LIN {X 0,Y 197.924,Z 366.595,A -85,B 0,C 180,E1 -22444.008,E2 -22444.008} C_VEL
LIN {X 0,Y 203.129,Z 358.179,A -85,B 0,C 180,E1 -22446.646,E2 -22446.646} C_VEL
LIN {X 0,Y 207.879,Z 349.395,A -85,B 0,C 180,E1 -22448.886,E2 -22448.886} C_VEL
LIN {X 0,Y 213.116,Z 339.014,A -85,B 0,C 180,E1 -22450.955,E2 -22450.955} C_VEL
LIN {X 0,Y 218.33,Z 327.013,A -85,B 0,C 180,E1 -22452.848,E2 -22452.848} C_VEL
LIN {X 0,Y 222.672,Z 315.199,A -85,B 0,C 180,E1 -22454.295,E2 -22454.295} C_VEL
LIN {X 0,Y 226.681,Z 302.215,A -85,B 0,C 180,E1 -22455.49,E2 -22455.49} C_VEL
LIN {X 0,Y 230.05,Z 288.122,A -85,B 0,C 180,E1 -22456.439,E2 -22456.439} C_VEL
LIN {X 0,Y 232.521,Z 273.354,A -85,B 0,C 180,E1 -22457.126,E2 -22457.126} C_VEL
LIN {X 0,Y 234.238,Z 254.152,A -85,B 0,C 180,E1 -22457.708,E2 -22457.708} C_VEL
LIN {X 0,Y 236.836,Z 218.214,A -85,B 0,C 180,E1 -22458.708,E2 -22458.708} C_VEL
LIN {X 0,Y 232.194,Z 207.283,A -85,B 0,C 180,E1 -22461.02,E2 -22461.02} C_VEL
LIN {X 0,Y 227.459,Z 197.713,A -85,B 0,C 180,E1 -22463.554,E2 -22463.554} C_VEL
LIN {X 0,Y 222.962,Z 189.346,A -85,B 0,C 180,E1 -22466.218,E2 -22466.218} C_VEL
LIN {X 0,Y 219.708,Z 183.706,A -85,B 0,C 180,E1 -22468.352,E2 -22468.352} C_VEL
LIN {X 0,Y 216.874,Z 179.005,A -85,B 0,C 180,E1 -22470.433,E2 -22470.433} C_VEL
LIN {X 0,Y 214.738,Z 175.538,A -85,B 0,C 180,E1 -22472.178,E2 -22472.178} C_VEL
LIN {X 0,Y 211.845,Z 170.966,A -85,B 0,C 180,E1 -22474.848,E2 -22474.848} C_VEL
LIN {X 0,Y 209.156,Z 167.545,A -85,B 0,C 180,E1 -22477.703,E2 -22477.703} C_VEL
LIN {X 0,Y 207.226,Z 164.238,A -85,B 0,C 180,E1 -22480.325,E2 -22480.325} C_VEL
LIN {X 0,Y 203.698,Z 160.294,A -85,B 0,C 180,E1 -22488.046,E2 -22488.046} C_VEL
LIN {X 0,Y 203.417,Z 158.582,A -85,B 0,C 180,E1 -22490.606,E2 -22490.606} C_VEL
LIN {X 0,Y 203.441,Z 158.596,A -85,B 0,C 180,E1 -22494.045,E2 -22494.045} C_VEL
LIN {X 0,Y 204.542,Z 161.074,A -85,B 0,C 180,E1 -22499.009,E2 -22499.009} C_VEL
LIN {X 0,Y 206.776,Z 163.712,A -85,B 0,C 180,E1 -22503.403,E2 -22503.403} C_VEL
LIN {X 0,Y 207.532,Z 164.297,A -85,B 0,C 180,E1 -22504.485,E2 -22504.485} C_VEL
LIN {X 0,Y 209.461,Z 167.504,A -85,B 0,C 180,E1 -22507.018,E2 -22507.018} C_VEL
LIN {X 0,Y 211.323,Z 169.48,A -85,B 0,C 180,E1 -22508.967,E2 -22508.967} C_VEL
LIN {X 0,Y 213.7,Z 172.996,A -85,B 0,C 180,E1 -22511.242,E2 -22511.242} C_VEL
LIN {X 0,Y 215.003,Z 174.469,A -85,B 0,C 180,E1 -22512.327,E2 -22512.327} C_VEL
LIN {X 0,Y 218.65,Z 179.753,A -85,B 0,C 180,E1 -22515.145,E2 -22515.145} C_VEL
LIN {X 0,Y 221.807,Z 184.294,A -85,B 0,C 180,E1 -22517.249,E2 -22517.249} C_VEL
LIN {X 0,Y 225.031,Z 189.073,A -85,B 0,C 180,E1 -22519.193,E2 -22519.193} C_VEL
LIN {X 0,Y 229.645,Z 196.427,A -85,B 0,C 180,E1 -22521.724,E2 -22521.724} C_VEL
LIN {X 0,Y 234.735,Z 206.452,A -85,B 0,C 180,E1 -22524.318,E2 -22524.318} C_VEL
LIN {X 0,Y 237.327,Z 212.29,A -85,B 0,C 180,E1 -22525.571,E2 -22525.571} C_VEL
LIN {X 0,Y 233.316,Z 263.334,A -85,B 0,C 180,E1 -22526.974,E2 -22526.974} C_VEL
LIN {X 0,Y 231.099,Z 278.043,A -85,B 0,C 180,E1 -22527.649,E2 -22527.649} C_VEL
LIN {X 0,Y 228.064,Z 291.816,A -85,B 0,C 180,E1 -22528.563,E2 -22528.563} C_VEL
LIN {X 0,Y 224.528,Z 304.669,A -85,B 0,C 180,E1 -22529.768,E2 -22529.768} C_VEL
LIN {X 0,Y 220.106,Z 317.534,A -85,B 0,C 180,E1 -22531.332,E2 -22531.332} C_VEL
LIN {X 0,Y 215.155,Z 329.395,A -85,B 0,C 180,E1 -22533.168,E2 -22533.168} C_VEL
LIN {X 0,Y 210.454,Z 339.175,A -85,B 0,C 180,E1 -22535.094,E2 -22535.094} C_VEL
LIN {X 0,Y 205.546,Z 348.318,A -85,B 0,C 180,E1 -22537.344,E2 -22537.344} C_VEL
LIN {X 0,Y 200.059,Z 357.453,A -85,B 0,C 180,E1 -22540.172,E2 -22540.172} C_VEL
LIN {X 0,Y 194.996,Z 365.083,A -85,B 0,C 180,E1 -22543.208,E2 -22543.208} C_VEL
LIN {X 0,Y 190,Z 372.03,A -85,B 0,C 180,E1 -22546.815,E2 -22546.815} C_VEL
LIN {X 0,Y 186.208,Z 376.82,A -85,B 0,C 180,E1 -22550.083,E2 -22550.083} C_VEL
LIN {X 0,Y 182.741,Z 380.951,A -85,B 0,C 180,E1 -22553.85,E2 -22553.85} C_VEL
LIN {X 0,Y 180.515,Z 383.439,A -85,B 0,C 180,E1 -22556.967,E2 -22556.967} C_VEL
LIN {X 0,Y 177.978,Z 385.836,A -85,B 0,C 180,E1 -22561.712,E2 -22561.712} C_VEL
LIN {X 0,Y 176.489,Z 386.756,A -85,B 0,C 180,E1 -22566.53,E2 -22566.53} C_VEL
LIN {X 0,Y 175.717,Z 386.244,A -85,B 0,C 180,E1 -22571.336,E2 -22571.336} C_VEL
LIN {X 0,Y 175.641,Z 385.441,A -85,B 0,C 180,E1 -22573.772,E2 -22573.772} C_VEL
LIN {X 0,Y 175.765,Z 382.819,A -85,B 0,C 180,E1 -22578.464,E2 -22578.464} C_VEL
LIN {X 0,Y 176.339,Z 379.84,A -85,B 0,C 180,E1 -22581.978,E2 -22581.978} C_VEL
LIN {X 0,Y 177.183,Z 376.025,A -85,B 0,C 180,E1 -22585.447,E2 -22585.447} C_VEL
LIN {X 0,Y 178.317,Z 371.31,A -85,B 0,C 180,E1 -22588.868,E2 -22588.868} C_VEL
LIN {X 0,Y 180.274,Z 364.443,A -85,B 0,C 180,E1 -22592.79,E2 -22592.79} C_VEL
LIN {X 0,Y 182.883,Z 355.918,A -85,B 0,C 180,E1 -22596.617,E2 -22596.617} C_VEL
LIN {X 0,Y 185.69,Z 346.926,A -85,B 0,C 180,E1 -22599.834,E2 -22599.834} C_VEL
LIN {X 0,Y 188.154,Z 338.243,A -85,B 0,C 180,E1 -22602.399,E2 -22602.399} C_VEL
LIN {X 0,Y 190.884,Z 328.903,A -85,B 0,C 180,E1 -22604.659,E2 -22604.659} C_VEL
LIN {X 0,Y 193.795,Z 317.727,A -85,B 0,C 180,E1 -22606.862,E2 -22606.862} C_VEL
LIN {X 0,Y 196.622,Z 305.546,A -85,B 0,C 180,E1 -22608.762,E2 -22608.762} C_VEL
LIN {X 0,Y 199.012,Z 293.194,A -85,B 0,C 180,E1 -22610.272,E2 -22610.272} C_VEL
LIN {X 0,Y 201.044,Z 279.549,A -85,B 0,C 180,E1 -22611.531,E2 -22611.531} C_VEL
LIN {X 0,Y 202.585,Z 265.477,A -85,B 0,C 180,E1 -22612.43,E2 -22612.43} C_VEL
LIN {X 0,Y 203.759,Z 246.646,A -85,B 0,C 180,E1 -22613.151,E2 -22613.151} C_VEL
LIN {X 0,Y 207.071,Z 187.142,A -85,B 0,C 180,E1 -22615.036,E2 -22615.036} C_VEL
LIN {X 0,Y 202.861,Z 176.015,A -85,B 0,C 180,E1 -22616.361,E2 -22616.361} C_VEL
LIN {X 0,Y 196.456,Z 163.46,A -85,B 0,C 180,E1 -22618.321,E2 -22618.321} C_VEL
LIN {X 0,Y 188.904,Z 150.475,A -85,B 0,C 180,E1 -22620.783,E2 -22620.783} C_VEL
LIN {X 0,Y 183.421,Z 142.139,A -85,B 0,C 180,E1 -22622.704,E2 -22622.704} C_VEL
LIN {X 0,Y 180.927,Z 138.404,A -85,B 0,C 180,E1 -22623.626,E2 -22623.626} C_VEL
LIN {X 0,Y 179.099,Z 136.063,A -85,B 0,C 180,E1 -22624.304,E2 -22624.304} C_VEL
LIN {X 0,Y 178.464,Z 133.88,A -85,B 0,C 180,E1 -22624.658,E2 -22624.658} C_VEL
LIN {X 0,Y 178.477,Z 133.875,A -85,B 0,C 180,E1 -22629.049,E2 -22629.049} C_VEL
LIN {X 0,Y 178.494,Z 133.859,A -85,B 0,C 180,E1 -22632.013,E2 -22632.013} C_VEL
LIN {X 0,Y 178.504,Z 133.854,A -85,B 0,C 180,E1 -22635.123,E2 -22635.123} C_VEL
LIN {X 0,Y 178.493,Z 133.87,A -85,B 0,C 180,E1 -22638.421,E2 -22638.421} C_VEL
LIN {X 0,Y 178.444,Z 133.86,A -85,B 0,C 180,E1 -22643.799,E2 -22643.799} C_VEL
LIN {X 0,Y 178.466,Z 133.878,A -85,B 0,C 180,E1 -22646.553,E2 -22646.553} C_VEL
LIN {X 0,Y 178.499,Z 133.842,A -85,B 0,C 180,E1 -22650.013,E2 -22650.013} C_VEL
LIN {X 0,Y 178.525,Z 133.862,A -85,B 0,C 180,E1 -22654.875,E2 -22654.875} C_VEL
LIN {X 0,Y 178.638,Z 133.852,A -85,B 0,C 180,E1 -22660.761,E2 -22660.761} C_VEL
LIN {X 0,Y 178.663,Z 133.849,A -85,B 0,C 180,E1 -22664.025,E2 -22664.025} C_VEL
LIN {X 0,Y 178.88,Z 133.825,A -85,B 0,C 180,E1 -22669.161,E2 -22669.161} C_VEL
LIN {X 0,Y 178.918,Z 133.782,A -85,B 0,C 180,E1 -22673.24,E2 -22673.24} C_VEL
LIN {X 0,Y 179.146,Z 133.788,A -85,B 0,C 180,E1 -22677.759,E2 -22677.759} C_VEL
LIN {X 0,Y 179.363,Z 133.764,A -85,B 0,C 180,E1 -22680.007,E2 -22680.007} C_VEL
LIN {X 0,Y 178.863,Z 133.791,A -85,B 0,C 180,E1 -22684.515,E2 -22684.515} C_VEL
LIN {X 0,Y 178.953,Z 133.817,A -85,B 0,C 180,E1 -22689.045,E2 -22689.045} C_VEL
LIN {X 0,Y 178.682,Z 133.85,A -85,B 0,C 180,E1 -22693.657,E2 -22693.657} C_VEL
LIN {X 0,Y 178.647,Z 133.853,A -85,B 0,C 180,E1 -22698.351,E2 -22698.351} C_VEL
LIN {X 0,Y 178.51,Z 133.872,A -85,B 0,C 180,E1 -22703.192,E2 -22703.192} C_VEL
LIN {X 0,Y 178.487,Z 133.863,A -85,B 0,C 180,E1 -22708.204,E2 -22708.204} C_VEL
LIN {X 0,Y 178.479,Z 133.872,A -85,B 0,C 180,E1 -22710.798,E2 -22710.798} C_VEL
LIN {X 0,Y 178.486,Z 133.875,A -85,B 0,C 180,E1 -22714.226,E2 -22714.226} C_VEL
LIN {X 0,Y 178.411,Z 134.02,A -85,B 0,C 180,E1 -22719,E2 -22719} C_VEL
LIN {X 0,Y 179.403,Z 136.688,A -85,B 0,C 180,E1 -22719.454,E2 -22719.454} C_VEL
LIN {X 0,Y 181.505,Z 139.246,A -85,B 0,C 180,E1 -22720.224,E2 -22720.224} C_VEL
LIN {X 0,Y 183.847,Z 142.743,A -85,B 0,C 180,E1 -22721.083,E2 -22721.083} C_VEL
LIN {X 0,Y 187.701,Z 149.384,A -85,B 0,C 180,E1 -22722.472,E2 -22722.472} C_VEL
LIN {X 0,Y 194.053,Z 161.878,A -85,B 0,C 180,E1 -22724.674,E2 -22724.674} C_VEL
LIN {X 0,Y 199.515,Z 174.348,A -85,B 0,C 180,E1 -22726.489,E2 -22726.489} C_VEL
LIN {X 0,Y 206.104,Z 192.069,A -85,B 0,C 180,E1 -22728.614,E2 -22728.614} C_VEL
LIN {X 0,Y 206.705,Z 198.43,A -85,B 0,C 180,E1 -22728.999,E2 -22728.999} C_VEL
LIN {X 0,Y 204.554,Z 239.005,A -85,B 0,C 180,E1 -22730.303,E2 -22730.303} C_VEL
LIN {X 0,Y 203.706,Z 244.85,A -85,B 0,C 180,E1 -22730.389,E2 -22730.389} C_VEL
LIN {X 0,Y 197.796,Z 263.79,A -85,B 0,C 180,E1 -22730.093,E2 -22730.093} C_VEL
LIN {X 0,Y 196.896,Z 269.616,A -85,B 0,C 180,E1 -22730.218,E2 -22730.218} C_VEL
LIN {X 0,Y 195.425,Z 283.938,A -85,B 0,C 180,E1 -22731.002,E2 -22731.002} C_VEL
LIN {X 0,Y 193.265,Z 297.901,A -85,B 0,C 180,E1 -22732.15,E2 -22732.15} C_VEL
LIN {X 0,Y 190.76,Z 310.487,A -85,B 0,C 180,E1 -22733.557,E2 -22733.557} C_VEL
LIN {X 0,Y 188.351,Z 320.636,A -85,B 0,C 180,E1 -22734.997,E2 -22734.997} C_VEL
LIN {X 0,Y 185.153,Z 333.155,A -85,B 0,C 180,E1 -22737.259,E2 -22737.259} C_VEL
LIN {X 0,Y 182.733,Z 341.231,A -85,B 0,C 180,E1 -22739.046,E2 -22739.046} C_VEL
LIN {X 0,Y 179.902,Z 350.234,A -85,B 0,C 180,E1 -22741.413,E2 -22741.413} C_VEL
LIN {X 0,Y 176.695,Z 360.281,A -85,B 0,C 180,E1 -22744.69,E2 -22744.69} C_VEL
LIN {X 0,Y 173.88,Z 369.292,A -85,B 0,C 180,E1 -22748.393,E2 -22748.393} C_VEL
LIN {X 0,Y 171.794,Z 376.544,A -85,B 0,C 180,E1 -22752.136,E2 -22752.136} C_VEL
LIN {X 0,Y 170.316,Z 382.067,A -85,B 0,C 180,E1 -22755.669,E2 -22755.669} C_VEL
LIN {X 0,Y 169.282,Z 387.851,A -85,B 0,C 180,E1 -22760.444,E2 -22760.444} C_VEL
LIN {X 0,Y 168.89,Z 392.01,A -85,B 0,C 180,E1 -22765.229,E2 -22765.229} C_VEL
LIN {X 0,Y 169.024,Z 394.686,A -85,B 0,C 180,E1 -22770.003,E2 -22770.003} C_VEL
LIN {X 0,Y 168.891,Z 395.944,A -85,B 0,C 180,E1 -22774.777,E2 -22774.777} C_VEL
LIN {X 0,Y 169.339,Z 395.878,A -85,B 0,C 180,E1 -22779.559,E2 -22779.559} C_VEL
LIN {X 0,Y 170.625,Z 394.512,A -85,B 0,C 180,E1 -22784.312,E2 -22784.312} C_VEL
LIN {X 0,Y 173.086,Z 391.826,A -85,B 0,C 180,E1 -22788.959,E2 -22788.959} C_VEL
LIN {X 0,Y 176.47,Z 387.752,A -85,B 0,C 180,E1 -22793.472,E2 -22793.472} C_VEL
LIN {X 0,Y 180.936,Z 382.174,A -85,B 0,C 180,E1 -22797.785,E2 -22797.785} C_VEL
LIN {X 0,Y 186.475,Z 374.921,A -85,B 0,C 180,E1 -22801.85,E2 -22801.85} C_VEL
LIN {X 0,Y 192.081,Z 366.957,A -85,B 0,C 180,E1 -22805.192,E2 -22805.192} C_VEL
LIN {X 0,Y 197.505,Z 358.65,A -85,B 0,C 180,E1 -22807.87,E2 -22807.87} C_VEL
LIN {X 0,Y 203.298,Z 348.508,A -85,B 0,C 180,E1 -22810.481,E2 -22810.481} C_VEL
LIN {X 0,Y 208.901,Z 337.643,A -85,B 0,C 180,E1 -22812.618,E2 -22812.618} C_VEL
LIN {X 0,Y 214.329,Z 325.298,A -85,B 0,C 180,E1 -22814.503,E2 -22814.503} C_VEL
LIN {X 0,Y 218.881,Z 313.11,A -85,B 0,C 180,E1 -22815.929,E2 -22815.929} C_VEL
LIN {X 0,Y 223.002,Z 299.6,A -85,B 0,C 180,E1 -22817.119,E2 -22817.119} C_VEL
LIN {X 0,Y 226.321,Z 285.451,A -85,B 0,C 180,E1 -22818.02,E2 -22818.02} C_VEL
LIN {X 0,Y 228.543,Z 271.735,A -85,B 0,C 180,E1 -22818.627,E2 -22818.627} C_VEL
LIN {X 0,Y 231.009,Z 242.939,A -85,B 0,C 180,E1 -22819.448,E2 -22819.448} C_VEL
LIN {X 0,Y 232.645,Z 221.01,A -85,B 0,C 180,E1 -22820.066,E2 -22820.066} C_VEL
LIN {X 0,Y 228.5,Z 211.213,A -85,B 0,C 180,E1 -22822.271,E2 -22822.271} C_VEL
LIN {X 0,Y 224.543,Z 202.944,A -85,B 0,C 180,E1 -22824.528,E2 -22824.528} C_VEL
LIN {X 0,Y 220.56,Z 195.258,A -85,B 0,C 180,E1 -22827.022,E2 -22827.022} C_VEL
LIN {X 0,Y 217.491,Z 189.717,A -85,B 0,C 180,E1 -22829.15,E2 -22829.15} C_VEL
LIN {X 0,Y 213.44,Z 182.601,A -85,B 0,C 180,E1 -22832.427,E2 -22832.427} C_VEL
LIN {X 0,Y 210.315,Z 177.667,A -85,B 0,C 180,E1 -22835.394,E2 -22835.394} C_VEL
LIN {X 0,Y 207.948,Z 174.459,A -85,B 0,C 180,E1 -22838.019,E2 -22838.019} C_VEL
LIN {X 0,Y 205.85,Z 170.917,A -85,B 0,C 180,E1 -22841.018,E2 -22841.018} C_VEL
LIN {X 0,Y 202.767,Z 167.321,A -85,B 0,C 180,E1 -22848.244,E2 -22848.244} C_VEL
LIN {X 0,Y 202.501,Z 165.535,A -85,B 0,C 180,E1 -22851.124,E2 -22851.124} C_VEL
LIN {X 0,Y 202.572,Z 165.825,A -85,B 0,C 180,E1 -22854.283,E2 -22854.283} C_VEL
LIN {X 0,Y 203.553,Z 168.062,A -85,B 0,C 180,E1 -22858.757,E2 -22858.757} C_VEL
LIN {X 0,Y 205.721,Z 170.676,A -85,B 0,C 180,E1 -22863.176,E2 -22863.176} C_VEL
LIN {X 0,Y 206.358,Z 171.324,A -85,B 0,C 180,E1 -22864.144,E2 -22864.144} C_VEL
LIN {X 0,Y 208.446,Z 174.671,A -85,B 0,C 180,E1 -22866.938,E2 -22866.938} C_VEL
LIN {X 0,Y 209.825,Z 176.191,A -85,B 0,C 180,E1 -22868.426,E2 -22868.426} C_VEL
LIN {X 0,Y 212.302,Z 179.809,A -85,B 0,C 180,E1 -22870.871,E2 -22870.871} C_VEL
LIN {X 0,Y 213.441,Z 181.322,A -85,B 0,C 180,E1 -22871.869,E2 -22871.869} C_VEL
LIN {X 0,Y 216.744,Z 186.164,A -85,B 0,C 180,E1 -22874.517,E2 -22874.517} C_VEL
LIN {X 0,Y 220.321,Z 191.498,A -85,B 0,C 180,E1 -22876.996,E2 -22876.996} C_VEL
LIN {X 0,Y 224.965,Z 198.794,A -85,B 0,C 180,E1 -22879.812,E2 -22879.812} C_VEL
LIN {X 0,Y 227.785,Z 203.912,A -85,B 0,C 180,E1 -22881.397,E2 -22881.397} C_VEL
LIN {X 0,Y 231.774,Z 212.095,A -85,B 0,C 180,E1 -22883.514,E2 -22883.514} C_VEL
LIN {X 0,Y 233.145,Z 215.09,A -85,B 0,C 180,E1 -22884.208,E2 -22884.208} C_VEL
LIN {X 0,Y 229.221,Z 263.339,A -85,B 0,C 180,E1 -22885.54,E2 -22885.54} C_VEL
LIN {X 0,Y 227.005,Z 277.668,A -85,B 0,C 180,E1 -22886.183,E2 -22886.183} C_VEL
LIN {X 0,Y 223.96,Z 291.248,A -85,B 0,C 180,E1 -22887.069,E2 -22887.069} C_VEL
LIN {X 0,Y 220.053,Z 304.97,A -85,B 0,C 180,E1 -22888.342,E2 -22888.342} C_VEL
LIN {X 0,Y 215.706,Z 317.209,A -85,B 0,C 180,E1 -22889.828,E2 -22889.828} C_VEL
LIN {X 0,Y 210.586,Z 329.163,A -85,B 0,C 180,E1 -22891.672,E2 -22891.672} C_VEL
LIN {X 0,Y 205.053,Z 340.237,A -85,B 0,C 180,E1 -22893.865,E2 -22893.865} C_VEL
LIN {X 0,Y 199.374,Z 350.201,A -85,B 0,C 180,E1 -22896.413,E2 -22896.413} C_VEL
LIN {X 0,Y 193.442,Z 359.417,A -85,B 0,C 180,E1 -22899.458,E2 -22899.458} C_VEL
LIN {X 0,Y 188.337,Z 366.604,A -85,B 0,C 180,E1 -22902.52,E2 -22902.52} C_VEL
LIN {X 0,Y 183.112,Z 373.348,A -85,B 0,C 180,E1 -22906.298,E2 -22906.298} C_VEL
LIN {X 0,Y 179.21,Z 377.935,A -85,B 0,C 180,E1 -22909.675,E2 -22909.675} C_VEL
LIN {X 0,Y 175.978,Z 381.516,A -85,B 0,C 180,E1 -22913.194,E2 -22913.194} C_VEL
LIN {X 0,Y 174.174,Z 383.378,A -85,B 0,C 180,E1 -22915.601,E2 -22915.601} C_VEL
LIN {X 0,Y 171.368,Z 385.895,A -85,B 0,C 180,E1 -22920.515,E2 -22920.515} C_VEL
LIN {X 0,Y 169.591,Z 386.933,A -85,B 0,C 180,E1 -22925.514,E2 -22925.514} C_VEL
LIN {X 0,Y 168.69,Z 386.534,A -85,B 0,C 180,E1 -22930.528,E2 -22930.528} C_VEL
LIN {X 0,Y 168.56,Z 385.64,A -85,B 0,C 180,E1 -22933.496,E2 -22933.496} C_VEL
LIN {X 0,Y 168.611,Z 383.286,A -85,B 0,C 180,E1 -22937.967,E2 -22937.967} C_VEL
LIN {X 0,Y 169.155,Z 380.413,A -85,B 0,C 180,E1 -22941.635,E2 -22941.635} C_VEL
LIN {X 0,Y 170.001,Z 376.719,A -85,B 0,C 180,E1 -22945.254,E2 -22945.254} C_VEL
LIN {X 0,Y 171.156,Z 372.089,A -85,B 0,C 180,E1 -22948.82,E2 -22948.82} C_VEL
LIN {X 0,Y 173.133,Z 365.392,A -85,B 0,C 180,E1 -22952.905,E2 -22952.905} C_VEL
LIN {X 0,Y 175.802,Z 357.048,A -85,B 0,C 180,E1 -22956.885,E2 -22956.885} C_VEL
LIN {X 0,Y 178.897,Z 347.578,A -85,B 0,C 180,E1 -22960.443,E2 -22960.443} C_VEL
LIN {X 0,Y 181.767,Z 337.828,A -85,B 0,C 180,E1 -22963.411,E2 -22963.411} C_VEL
LIN {X 0,Y 184.659,Z 328.358,A -85,B 0,C 180,E1 -22965.731,E2 -22965.731} C_VEL
LIN {X 0,Y 187.723,Z 317.019,A -85,B 0,C 180,E1 -22967.988,E2 -22967.988} C_VEL
LIN {X 0,Y 190.645,Z 304.637,A -85,B 0,C 180,E1 -22969.934,E2 -22969.934} C_VEL
LIN {X 0,Y 193.38,Z 290.832,A -85,B 0,C 180,E1 -22971.587,E2 -22971.587} C_VEL
LIN {X 0,Y 195.342,Z 277.108,A -85,B 0,C 180,E1 -22972.82,E2 -22972.82} C_VEL
LIN {X 0,Y 196.867,Z 262.852,A -85,B 0,C 180,E1 -22973.677,E2 -22973.677} C_VEL
LIN {X 0,Y 200.885,Z 196.744,A -85,B 0,C 180,E1 -22975.858,E2 -22975.858} C_VEL
LIN {X 0,Y 201.212,Z 188.949,A -85,B 0,C 180,E1 -22976.135,E2 -22976.135} C_VEL
LIN {X 0,Y 197.357,Z 178.875,A -85,B 0,C 180,E1 -22977.409,E2 -22977.409} C_VEL
LIN {X 0,Y 191.075,Z 166.594,A -85,B 0,C 180,E1 -22979.443,E2 -22979.443} C_VEL
LIN {X 0,Y 184.097,Z 154.645,A -85,B 0,C 180,E1 -22981.856,E2 -22981.856} C_VEL
LIN {X 0,Y 177.132,Z 143.849,A -85,B 0,C 180,E1 -22984.475,E2 -22984.475} C_VEL
LIN {X 0,Y 174.957,Z 140.891,A -85,B 0,C 180,E1 -22985.334,E2 -22985.334} C_VEL
LIN {X 0,Y 174.114,Z 139.492,A -85,B 0,C 180,E1 -22985.691,E2 -22985.691} C_VEL
LIN {X 0,Y 172.15,Z 137.141,A -85,B 0,C 180,E1 -22986.492,E2 -22986.492} C_VEL
LIN {X 0,Y 171.41,Z 134.76,A -85,B 0,C 180,E1 -22986.954,E2 -22986.954} C_VEL
LIN {X 0,Y 171.434,Z 134.733,A -85,B 0,C 180,E1 -22992.46,E2 -22992.46} C_VEL
LIN {X 0,Y 171.432,Z 134.753,A -85,B 0,C 180,E1 -22997.549,E2 -22997.549} C_VEL
LIN {X 0,Y 171.417,Z 134.721,A -85,B 0,C 180,E1 -23002.06,E2 -23002.06} C_VEL
LIN {X 0,Y 171.395,Z 134.752,A -85,B 0,C 180,E1 -23007.798,E2 -23007.798} C_VEL
LIN {X 0,Y 171.426,Z 134.718,A -85,B 0,C 180,E1 -23010.54,E2 -23010.54} C_VEL
LIN {X 0,Y 171.453,Z 134.75,A -85,B 0,C 180,E1 -23015.81,E2 -23015.81} C_VEL
LIN {X 0,Y 171.594,Z 134.73,A -85,B 0,C 180,E1 -23020.882,E2 -23020.882} C_VEL
LIN {X 0,Y 171.599,Z 134.724,A -85,B 0,C 180,E1 -23025.783,E2 -23025.783} C_VEL
LIN {X 0,Y 171.894,Z 134.682,A -85,B 0,C 180,E1 -23030.596,E2 -23030.596} C_VEL
LIN {X 0,Y 171.814,Z 134.673,A -85,B 0,C 180,E1 -23035.315,E2 -23035.315} C_VEL
LIN {X 0,Y 172.325,Z 134.641,A -85,B 0,C 180,E1 -23040.008,E2 -23040.008} C_VEL
LIN {X 0,Y 171.812,Z 134.668,A -85,B 0,C 180,E1 -23044.7,E2 -23044.7} C_VEL
LIN {X 0,Y 171.883,Z 134.7,A -85,B 0,C 180,E1 -23049.421,E2 -23049.421} C_VEL
LIN {X 0,Y 171.605,Z 134.733,A -85,B 0,C 180,E1 -23054.232,E2 -23054.232} C_VEL
LIN {X 0,Y 171.542,Z 134.742,A -85,B 0,C 180,E1 -23059.57,E2 -23059.57} C_VEL
LIN {X 0,Y 171.469,Z 134.749,A -85,B 0,C 180,E1 -23065.624,E2 -23065.624} C_VEL
LIN {X 0,Y 171.442,Z 134.75,A -85,B 0,C 180,E1 -23070.594,E2 -23070.594} C_VEL
LIN {X 0,Y 171.391,Z 134.759,A -85,B 0,C 180,E1 -23076.674,E2 -23076.674} C_VEL
LIN {X 0,Y 172.273,Z 137.408,A -85,B 0,C 180,E1 -23077.185,E2 -23077.185} C_VEL
LIN {X 0,Y 174.601,Z 140.281,A -85,B 0,C 180,E1 -23078.138,E2 -23078.138} C_VEL
LIN {X 0,Y 176.859,Z 143.654,A -85,B 0,C 180,E1 -23079.056,E2 -23079.056} C_VEL
LIN {X 0,Y 181.273,Z 150.337,A -85,B 0,C 180,E1 -23080.752,E2 -23080.752} C_VEL
LIN {X 0,Y 187.224,Z 161.787,A -85,B 0,C 180,E1 -23082.972,E2 -23082.972} C_VEL
LIN {X 0,Y 193.134,Z 174.722,A -85,B 0,C 180,E1 -23085.065,E2 -23085.065} C_VEL
LIN {X 0,Y 199.773,Z 192.505,A -85,B 0,C 180,E1 -23087.355,E2 -23087.355} C_VEL
LIN {X 0,Y 200.578,Z 195.555,A -85,B 0,C 180,E1 -23087.658,E2 -23087.658} C_VEL
LIN {X 0,Y 200.842,Z 199.819,A -85,B 0,C 180,E1 -23087.9,E2 -23087.9} C_VEL
LIN {X 0,Y 196.896,Z 269.616,A -85,B 0,C 180,E1 -23090.218,E2 -23090.218} C_VEL
LIN {X 0,Y 195.922,Z 275.406,A -85,B 0,C 180,E1 -23090.387,E2 -23090.387} C_VEL
LIN {X 0,Y 192.489,Z 284.69,A -85,B 0,C 180,E1 -23090.5,E2 -23090.5} C_VEL
LIN {X 0,Y 188.597,Z 293.797,A -85,B 0,C 180,E1 -23090.762,E2 -23090.762} C_VEL
LIN {X 0,Y 186.917,Z 299.319,A -85,B 0,C 180,E1 -23091.172,E2 -23091.172} C_VEL
LIN {X 0,Y 184.148,Z 312.294,A -85,B 0,C 180,E1 -23092.713,E2 -23092.713} C_VEL
LIN {X 0,Y 181.138,Z 324.295,A -85,B 0,C 180,E1 -23094.576,E2 -23094.576} C_VEL
LIN {X 0,Y 178.365,Z 334.301,A -85,B 0,C 180,E1 -23096.525,E2 -23096.525} C_VEL
LIN {X 0,Y 175.977,Z 342.273,A -85,B 0,C 180,E1 -23098.391,E2 -23098.391} C_VEL
LIN {X 0,Y 172.398,Z 352.871,A -85,B 0,C 180,E1 -23101.384,E2 -23101.384} C_VEL
LIN {X 0,Y 169.237,Z 362.449,A -85,B 0,C 180,E1 -23104.812,E2 -23104.812} C_VEL
LIN {X 0,Y 166.629,Z 370.348,A -85,B 0,C 180,E1 -23108.338,E2 -23108.338} C_VEL
LIN {X 0,Y 164.425,Z 377.927,A -85,B 0,C 180,E1 -23112.594,E2 -23112.594} C_VEL
LIN {X 0,Y 163.006,Z 383.156,A -85,B 0,C 180,E1 -23116.286,E2 -23116.286} C_VEL
LIN {X 0,Y 162.227,Z 387.382,A -85,B 0,C 180,E1 -23120.025,E2 -23120.025} C_VEL
LIN {X 0,Y 161.946,Z 389.695,A -85,B 0,C 180,E1 -23122.523,E2 -23122.523} C_VEL
LIN {X 0,Y 161.814,Z 393.172,A -85,B 0,C 180,E1 -23127.514,E2 -23127.514} C_VEL
LIN {X 0,Y 161.934,Z 394.368,A -85,B 0,C 180,E1 -23130.004,E2 -23130.004} C_VEL
LIN {X 0,Y 161.81,Z 395.698,A -85,B 0,C 180,E1 -23134.987,E2 -23134.987} C_VEL
LIN {X 0,Y 162.326,Z 395.706,A -85,B 0,C 180,E1 -23139.976,E2 -23139.976} C_VEL
LIN {X 0,Y 163.709,Z 394.42,A -85,B 0,C 180,E1 -23144.93,E2 -23144.93} C_VEL
LIN {X 0,Y 166.338,Z 391.824,A -85,B 0,C 180,E1 -23149.759,E2 -23149.759} C_VEL
LIN {X 0,Y 169.94,Z 387.837,A -85,B 0,C 180,E1 -23154.432,E2 -23154.432} C_VEL
LIN {X 0,Y 174.677,Z 382.342,A -85,B 0,C 180,E1 -23158.873,E2 -23158.873} C_VEL
LIN {X 0,Y 180.486,Z 375.178,A -85,B 0,C 180,E1 -23163.038,E2 -23163.038} C_VEL
LIN {X 0,Y 186.339,Z 367.314,A -85,B 0,C 180,E1 -23166.447,E2 -23166.447} C_VEL
LIN {X 0,Y 191.977,Z 359.12,A -85,B 0,C 180,E1 -23169.164,E2 -23169.164} C_VEL
LIN {X 0,Y 197.774,Z 349.473,A -85,B 0,C 180,E1 -23171.726,E2 -23171.726} C_VEL
LIN {X 0,Y 203.783,Z 338.448,A -85,B 0,C 180,E1 -23173.956,E2 -23173.956} C_VEL
LIN {X 0,Y 209.379,Z 326.422,A -85,B 0,C 180,E1 -23175.85,E2 -23175.85} C_VEL
LIN {X 0,Y 214.066,Z 314.565,A -85,B 0,C 180,E1 -23177.276,E2 -23177.276} C_VEL
LIN {X 0,Y 218.601,Z 300.415,A -85,B 0,C 180,E1 -23178.55,E2 -23178.55} C_VEL
LIN {X 0,Y 222.027,Z 286.604,A -85,B 0,C 180,E1 -23179.44,E2 -23179.44} C_VEL
LIN {X 0,Y 224.423,Z 272.754,A -85,B 0,C 180,E1 -23180.072,E2 -23180.072} C_VEL
LIN {X 0,Y 226.373,Z 252.123,A -85,B 0,C 180,E1 -23180.688,E2 -23180.688} C_VEL
LIN {X 0,Y 228.588,Z 223.962,A -85,B 0,C 180,E1 -23181.469,E2 -23181.469} C_VEL
LIN {X 0,Y 225.133,Z 215.618,A -85,B 0,C 180,E1 -23183.437,E2 -23183.437} C_VEL
LIN {X 0,Y 221.106,Z 206.893,A -85,B 0,C 180,E1 -23185.908,E2 -23185.908} C_VEL
LIN {X 0,Y 217.495,Z 199.828,A -85,B 0,C 180,E1 -23188.341,E2 -23188.341} C_VEL
LIN {X 0,Y 213.873,Z 193.038,A -85,B 0,C 180,E1 -23191.153,E2 -23191.153} C_VEL
LIN {X 0,Y 211.177,Z 188.352,A -85,B 0,C 180,E1 -23193.54,E2 -23193.54} C_VEL
LIN {X 0,Y 208.172,Z 183.358,A -85,B 0,C 180,E1 -23196.654,E2 -23196.654} C_VEL
LIN {X 0,Y 204.661,Z 177.829,A -85,B 0,C 180,E1 -23201.448,E2 -23201.448} C_VEL
LIN {X 0,Y 201.755,Z 174.043,A -85,B 0,C 180,E1 -23208.948,E2 -23208.948} C_VEL
LIN {X 0,Y 201.611,Z 172.649,A -85,B 0,C 180,E1 -23211.085,E2 -23211.085} C_VEL
LIN {X 0,Y 201.658,Z 172.794,A -85,B 0,C 180,E1 -23213.992,E2 -23213.992} C_VEL
LIN {X 0,Y 202.581,Z 175.069,A -85,B 0,C 180,E1 -23218.548,E2 -23218.548} C_VEL
LIN {X 0,Y 204.668,Z 177.649,A -85,B 0,C 180,E1 -23222.946,E2 -23222.946} C_VEL
LIN {X 0,Y 205.196,Z 178.331,A -85,B 0,C 180,E1 -23223.798,E2 -23223.798} C_VEL
LIN {X 0,Y 207.332,Z 181.654,A -85,B 0,C 180,E1 -23226.731,E2 -23226.731} C_VEL
LIN {X 0,Y 208.445,Z 183.081,A -85,B 0,C 180,E1 -23227.99,E2 -23227.99} C_VEL
LIN {X 0,Y 211.139,Z 186.884,A -85,B 0,C 180,E1 -23230.699,E2 -23230.699} C_VEL
LIN {X 0,Y 214.806,Z 192.528,A -85,B 0,C 180,E1 -23233.835,E2 -23233.835} C_VEL
LIN {X 0,Y 219.154,Z 199.151,A -85,B 0,C 180,E1 -23236.943,E2 -23236.943} C_VEL
LIN {X 0,Y 224.114,Z 207.619,A -85,B 0,C 180,E1 -23240.003,E2 -23240.003} C_VEL
LIN {X 0,Y 228.412,Z 216.669,A -85,B 0,C 180,E1 -23242.442,E2 -23242.442} C_VEL
LIN {X 0,Y 229.075,Z 218.347,A -85,B 0,C 180,E1 -23242.812,E2 -23242.812} C_VEL
LIN {X 0,Y 225.192,Z 264.021,A -85,B 0,C 180,E1 -23244.078,E2 -23244.078} C_VEL
LIN {X 0,Y 222.852,Z 278.551,A -85,B 0,C 180,E1 -23244.743,E2 -23244.743} C_VEL
LIN {X 0,Y 219.706,Z 291.942,A -85,B 0,C 180,E1 -23245.616,E2 -23245.616} C_VEL
LIN {X 0,Y 215.634,Z 305.657,A -85,B 0,C 180,E1 -23246.895,E2 -23246.895} C_VEL
LIN {X 0,Y 210.871,Z 318.464,A -85,B 0,C 180,E1 -23248.469,E2 -23248.469} C_VEL
LIN {X 0,Y 205.578,Z 330.204,A -85,B 0,C 180,E1 -23250.316,E2 -23250.316} C_VEL
LIN {X 0,Y 199.962,Z 340.898,A -85,B 0,C 180,E1 -23252.482,E2 -23252.482} C_VEL
LIN {X 0,Y 193.906,Z 350.983,A -85,B 0,C 180,E1 -23255.118,E2 -23255.118} C_VEL
LIN {X 0,Y 187.778,Z 360.033,A -85,B 0,C 180,E1 -23258.185,E2 -23258.185} C_VEL
LIN {X 0,Y 182.167,Z 367.493,A -85,B 0,C 180,E1 -23261.482,E2 -23261.482} C_VEL
LIN {X 0,Y 176.666,Z 374.155,A -85,B 0,C 180,E1 -23265.397,E2 -23265.397} C_VEL
LIN {X 0,Y 172.236,Z 378.99,A -85,B 0,C 180,E1 -23269.237,E2 -23269.237} C_VEL
LIN {X 0,Y 169.814,Z 381.493,A -85,B 0,C 180,E1 -23271.83,E2 -23271.83} C_VEL
LIN {X 0,Y 166.267,Z 384.817,A -85,B 0,C 180,E1 -23276.663,E2 -23276.663} C_VEL
LIN {X 0,Y 163.651,Z 386.716,A -85,B 0,C 180,E1 -23281.806,E2 -23281.806} C_VEL
LIN {X 0,Y 162.113,Z 387.145,A -85,B 0,C 180,E1 -23287.031,E2 -23287.031} C_VEL
LIN {X 0,Y 161.478,Z 386.148,A -85,B 0,C 180,E1 -23292.259,E2 -23292.259} C_VEL
LIN {X 0,Y 161.414,Z 385.121,A -85,B 0,C 180,E1 -23294.853,E2 -23294.853} C_VEL
LIN {X 0,Y 161.769,Z 382.001,A -85,B 0,C 180,E1 -23299.989,E2 -23299.989} C_VEL
LIN {X 0,Y 162.538,Z 378.564,A -85,B 0,C 180,E1 -23303.893,E2 -23303.893} C_VEL
LIN {X 0,Y 163.976,Z 372.847,A -85,B 0,C 180,E1 -23308.769,E2 -23308.769} C_VEL
LIN {X 0,Y 165.978,Z 366.288,A -85,B 0,C 180,E1 -23313.031,E2 -23313.031} C_VEL
LIN {X 0,Y 168.723,Z 358.15,A -85,B 0,C 180,E1 -23317.175,E2 -23317.175} C_VEL
LIN {X 0,Y 171.458,Z 350.198,A -85,B 0,C 180,E1 -23320.396,E2 -23320.396} C_VEL
LIN {X 0,Y 174.337,Z 341.181,A -85,B 0,C 180,E1 -23323.399,E2 -23323.399} C_VEL
LIN {X 0,Y 177.381,Z 331.208,A -85,B 0,C 180,E1 -23326.098,E2 -23326.098} C_VEL
LIN {X 0,Y 180.595,Z 320.4,A -85,B 0,C 180,E1 -23328.429,E2 -23328.429} C_VEL
LIN {X 0,Y 183.593,Z 308.772,A -85,B 0,C 180,E1 -23330.441,E2 -23330.441} C_VEL
LIN {X 0,Y 186.561,Z 295.143,A -85,B 0,C 180,E1 -23332.273,E2 -23332.273} C_VEL
LIN {X 0,Y 188.767,Z 282.077,A -85,B 0,C 180,E1 -23333.589,E2 -23333.589} C_VEL
LIN {X 0,Y 190.472,Z 268.076,A -85,B 0,C 180,E1 -23334.595,E2 -23334.595} C_VEL
LIN {X 0,Y 191.688,Z 253.405,A -85,B 0,C 180,E1 -23335.224,E2 -23335.224} C_VEL
LIN {X 0,Y 195.398,Z 190.619,A -85,B 0,C 180,E1 -23337.304,E2 -23337.304} C_VEL
LIN {X 0,Y 192.258,Z 182.569,A -85,B 0,C 180,E1 -23338.394,E2 -23338.394} C_VEL
LIN {X 0,Y 186.411,Z 170.947,A -85,B 0,C 180,E1 -23340.402,E2 -23340.402} C_VEL
LIN {X 0,Y 179.803,Z 159.387,A -85,B 0,C 180,E1 -23342.819,E2 -23342.819} C_VEL
LIN {X 0,Y 173.098,Z 148.974,A -85,B 0,C 180,E1 -23345.472,E2 -23345.472} C_VEL
LIN {X 0,Y 169.895,Z 144.445,A -85,B 0,C 180,E1 -23346.833,E2 -23346.833} C_VEL
LIN {X 0,Y 167.685,Z 140.987,A -85,B 0,C 180,E1 -23347.845,E2 -23347.845} C_VEL
LIN {X 0,Y 165.205,Z 138.17,A -85,B 0,C 180,E1 -23348.967,E2 -23348.967} C_VEL
LIN {X 0,Y 164.377,Z 135.633,A -85,B 0,C 180,E1 -23349.532,E2 -23349.532} C_VEL
LIN {X 0,Y 164.367,Z 135.607,A -85,B 0,C 180,E1 -23353.388,E2 -23353.388} C_VEL
LIN {X 0,Y 164.371,Z 135.63,A -85,B 0,C 180,E1 -23356.847,E2 -23356.847} C_VEL
LIN {X 0,Y 164.352,Z 135.607,A -85,B 0,C 180,E1 -23360.322,E2 -23360.322} C_VEL
LIN {X 0,Y 164.324,Z 135.623,A -85,B 0,C 180,E1 -23364.346,E2 -23364.346} C_VEL
LIN {X 0,Y 164.367,Z 135.61,A -85,B 0,C 180,E1 -23369.14,E2 -23369.14} C_VEL
LIN {X 0,Y 164.404,Z 135.617,A -85,B 0,C 180,E1 -23374.702,E2 -23374.702} C_VEL
LIN {X 0,Y 164.502,Z 135.609,A -85,B 0,C 180,E1 -23380.024,E2 -23380.024} C_VEL
LIN {X 0,Y 164.546,Z 135.602,A -85,B 0,C 180,E1 -23385.16,E2 -23385.16} C_VEL
LIN {X 0,Y 164.837,Z 135.565,A -85,B 0,C 180,E1 -23390.189,E2 -23390.189} C_VEL
LIN {X 0,Y 164.763,Z 135.547,A -85,B 0,C 180,E1 -23395.114,E2 -23395.114} C_VEL
LIN {X 0,Y 165.287,Z 135.518,A -85,B 0,C 180,E1 -23400.008,E2 -23400.008} C_VEL
LIN {X 0,Y 164.762,Z 135.545,A -85,B 0,C 180,E1 -23404.902,E2 -23404.902} C_VEL
LIN {X 0,Y 164.844,Z 135.558,A -85,B 0,C 180,E1 -23407.356,E2 -23407.356} C_VEL
LIN {X 0,Y 164.748,Z 135.583,A -85,B 0,C 180,E1 -23411.16,E2 -23411.16} C_VEL
LIN {X 0,Y 164.502,Z 135.611,A -85,B 0,C 180,E1 -23417.409,E2 -23417.409} C_VEL
LIN {X 0,Y 164.471,Z 135.623,A -85,B 0,C 180,E1 -23419.997,E2 -23419.997} C_VEL
LIN {X 0,Y 164.393,Z 135.626,A -85,B 0,C 180,E1 -23426.142,E2 -23426.142} C_VEL
LIN {X 0,Y 164.376,Z 135.626,A -85,B 0,C 180,E1 -23431.235,E2 -23431.235} C_VEL
LIN {X 0,Y 164.334,Z 135.731,A -85,B 0,C 180,E1 -23434.147,E2 -23434.147} C_VEL
LIN {X 0,Y 165.151,Z 138.154,A -85,B 0,C 180,E1 -23434.626,E2 -23434.626} C_VEL
LIN {X 0,Y 167.212,Z 140.507,A -85,B 0,C 180,E1 -23435.563,E2 -23435.563} C_VEL
LIN {X 0,Y 170.151,Z 144.786,A -85,B 0,C 180,E1 -23436.893,E2 -23436.893} C_VEL
LIN {X 0,Y 176.242,Z 153.813,A -85,B 0,C 180,E1 -23439.436,E2 -23439.436} C_VEL
LIN {X 0,Y 179.678,Z 160.01,A -85,B 0,C 180,E1 -23440.811,E2 -23440.811} C_VEL
LIN {X 0,Y 186.476,Z 174.512,A -85,B 0,C 180,E1 -23443.419,E2 -23443.419} C_VEL
LIN {X 0,Y 191.641,Z 187.698,A -85,B 0,C 180,E1 -23445.33,E2 -23445.33} C_VEL
LIN {X 0,Y 194.915,Z 197.202,A -85,B 0,C 180,E1 -23446.522,E2 -23446.522} C_VEL
LIN {X 0,Y 195.059,Z 200.705,A -85,B 0,C 180,E1 -23446.714,E2 -23446.714} C_VEL
LIN {X 0,Y 190.913,Z 271.053,A -85,B 0,C 180,E1 -23449.117,E2 -23449.117} C_VEL
LIN {X 0,Y 189.219,Z 285.687,A -85,B 0,C 180,E1 -23449.987,E2 -23449.987} C_VEL
LIN {X 0,Y 186.96,Z 299.125,A -85,B 0,C 180,E1 -23451.153,E2 -23451.153} C_VEL
LIN {X 0,Y 186.917,Z 299.319,A -85,B 0,C 180,E1 -23451.172,E2 -23451.172} C_VEL
LIN {X 0,Y 185.154,Z 304.813,A -85,B 0,C 180,E1 -23451.642,E2 -23451.642} C_VEL
LIN {X 0,Y 180.723,Z 313.415,A -85,B 0,C 180,E1 -23452.28,E2 -23452.28} C_VEL
LIN {X 0,Y 176.177,Z 321.783,A -85,B 0,C 180,E1 -23453.133,E2 -23453.133} C_VEL
LIN {X 0,Y 174.269,Z 326.771,A -85,B 0,C 180,E1 -23453.944,E2 -23453.944} C_VEL
LIN {X 0,Y 171.2,Z 336.589,A -85,B 0,C 180,E1 -23455.995,E2 -23455.995} C_VEL
LIN {X 0,Y 168.186,Z 346.259,A -85,B 0,C 180,E1 -23458.515,E2 -23458.515} C_VEL
LIN {X 0,Y 164.935,Z 355.301,A -85,B 0,C 180,E1 -23461.36,E2 -23461.36} C_VEL
LIN {X 0,Y 161.773,Z 364.409,A -85,B 0,C 180,E1 -23464.944,E2 -23464.944} C_VEL
LIN {X 0,Y 159.266,Z 371.711,A -85,B 0,C 180,E1 -23468.505,E2 -23468.505} C_VEL
LIN {X 0,Y 157.613,Z 377.307,A -85,B 0,C 180,E1 -23471.816,E2 -23471.816} C_VEL
LIN {X 0,Y 156.049,Z 382.598,A -85,B 0,C 180,E1 -23475.662,E2 -23475.662} C_VEL
LIN {X 0,Y 155.032,Z 388.168,A -85,B 0,C 180,E1 -23480.874,E2 -23480.874} C_VEL
LIN {X 0,Y 154.724,Z 391.226,A -85,B 0,C 180,E1 -23484.792,E2 -23484.792} C_VEL
LIN {X 0,Y 154.729,Z 393.142,A -85,B 0,C 180,E1 -23487.987,E2 -23487.987} C_VEL
LIN {X 0,Y 154.835,Z 394.047,A -85,B 0,C 180,E1 -23490.004,E2 -23490.004} C_VEL
LIN {X 0,Y 154.725,Z 395.448,A -85,B 0,C 180,E1 -23495.216,E2 -23495.216} C_VEL
LIN {X 0,Y 155.298,Z 395.527,A -85,B 0,C 180,E1 -23500.433,E2 -23500.433} C_VEL
LIN {X 0,Y 156.816,Z 394.313,A -85,B 0,C 180,E1 -23505.603,E2 -23505.603} C_VEL
LIN {X 0,Y 159.628,Z 391.797,A -85,B 0,C 180,E1 -23510.627,E2 -23510.627} C_VEL
LIN {X 0,Y 163.487,Z 387.911,A -85,B 0,C 180,E1 -23515.464,E2 -23515.464} C_VEL
LIN {X 0,Y 168.471,Z 382.51,A -85,B 0,C 180,E1 -23520.043,E2 -23520.043} C_VEL
LIN {X 0,Y 174.566,Z 375.443,A -85,B 0,C 180,E1 -23524.311,E2 -23524.311} C_VEL
LIN {X 0,Y 180.698,Z 367.692,A -85,B 0,C 180,E1 -23527.78,E2 -23527.78} C_VEL
LIN {X 0,Y 186.552,Z 359.628,A -85,B 0,C 180,E1 -23530.535,E2 -23530.535} C_VEL
LIN {X 0,Y 192.865,Z 349.635,A -85,B 0,C 180,E1 -23533.237,E2 -23533.237} C_VEL
LIN {X 0,Y 199.33,Z 338.208,A -85,B 0,C 180,E1 -23535.563,E2 -23535.563} C_VEL
LIN {X 0,Y 205.116,Z 326.173,A -85,B 0,C 180,E1 -23537.452,E2 -23537.452} C_VEL
LIN {X 0,Y 209.986,Z 314.294,A -85,B 0,C 180,E1 -23538.859,E2 -23538.859} C_VEL
LIN {X 0,Y 214.659,Z 300.117,A -85,B 0,C 180,E1 -23540.12,E2 -23540.12} C_VEL
LIN {X 0,Y 218.338,Z 285.564,A -85,B 0,C 180,E1 -23541.036,E2 -23541.036} C_VEL
LIN {X 0,Y 220.673,Z 272.137,A -85,B 0,C 180,E1 -23541.634,E2 -23541.634} C_VEL
LIN {X 0,Y 222.743,Z 250.64,A -85,B 0,C 180,E1 -23542.263,E2 -23542.263} C_VEL
LIN {X 0,Y 224.69,Z 226.904,A -85,B 0,C 180,E1 -23542.915,E2 -23542.915} C_VEL
LIN {X 0,Y 220.725,Z 217.299,A -85,B 0,C 180,E1 -23545.369,E2 -23545.369} C_VEL
LIN {X 0,Y 216.281,Z 207.768,A -85,B 0,C 180,E1 -23548.405,E2 -23548.405} C_VEL
LIN {X 0,Y 212.147,Z 199.622,A -85,B 0,C 180,E1 -23551.726,E2 -23551.726} C_VEL
LIN {X 0,Y 209.361,Z 194.613,A -85,B 0,C 180,E1 -23554.321,E2 -23554.321} C_VEL
LIN {X 0,Y 206.557,Z 189.777,A -85,B 0,C 180,E1 -23557.407,E2 -23557.407} C_VEL
LIN {X 0,Y 203.483,Z 184.732,A -85,B 0,C 180,E1 -23561.884,E2 -23561.884} C_VEL
LIN {X 0,Y 200.773,Z 180.763,A -85,B 0,C 180,E1 -23569.659,E2 -23569.659} C_VEL
LIN {X 0,Y 200.704,Z 179.643,A -85,B 0,C 180,E1 -23571.493,E2 -23571.493} C_VEL
LIN {X 0,Y 200.759,Z 179.928,A -85,B 0,C 180,E1 -23573.965,E2 -23573.965} C_VEL
LIN {X 0,Y 201.566,Z 181.948,A -85,B 0,C 180,E1 -23578.177,E2 -23578.177} C_VEL
LIN {X 0,Y 203.62,Z 184.599,A -85,B 0,C 180,E1 -23582.712,E2 -23582.712} C_VEL
LIN {X 0,Y 206.528,Z 189.013,A -85,B 0,C 180,E1 -23586.886,E2 -23586.886} C_VEL
LIN {X 0,Y 210.239,Z 194.669,A -85,B 0,C 180,E1 -23590.804,E2 -23590.804} C_VEL
LIN {X 0,Y 213.207,Z 199.393,A -85,B 0,C 180,E1 -23593.395,E2 -23593.395} C_VEL
LIN {X 0,Y 216.076,Z 203.955,A -85,B 0,C 180,E1 -23595.589,E2 -23595.589} C_VEL
LIN {X 0,Y 220.486,Z 211.41,A -85,B 0,C 180,E1 -23598.523,E2 -23598.523} C_VEL
LIN {X 0,Y 224.794,Z 220.413,A -85,B 0,C 180,E1 -23601.139,E2 -23601.139} C_VEL
LIN {X 0,Y 225.14,Z 221.282,A -85,B 0,C 180,E1 -23601.345,E2 -23601.345} C_VEL
LIN {X 0,Y 221.364,Z 264.336,A -85,B 0,C 180,E1 -23602.548,E2 -23602.548} C_VEL
LIN {X 0,Y 218.988,Z 278.605,A -85,B 0,C 180,E1 -23603.19,E2 -23603.19} C_VEL
LIN {X 0,Y 215.597,Z 292.636,A -85,B 0,C 180,E1 -23604.108,E2 -23604.108} C_VEL
LIN {X 0,Y 211.778,Z 305.121,A -85,B 0,C 180,E1 -23605.264,E2 -23605.264} C_VEL
LIN {X 0,Y 206.714,Z 318.373,A -85,B 0,C 180,E1 -23606.865,E2 -23606.865} C_VEL
LIN {X 0,Y 201.299,Z 330.048,A -85,B 0,C 180,E1 -23608.689,E2 -23608.689} C_VEL
LIN {X 0,Y 196.006,Z 339.795,A -85,B 0,C 180,E1 -23610.617,E2 -23610.617} C_VEL
LIN {X 0,Y 190.464,Z 348.922,A -85,B 0,C 180,E1 -23612.913,E2 -23612.913} C_VEL
LIN {X 0,Y 184.173,Z 358.034,A -85,B 0,C 180,E1 -23615.812,E2 -23615.812} C_VEL
LIN {X 0,Y 178.039,Z 366.025,A -85,B 0,C 180,E1 -23619.157,E2 -23619.157} C_VEL
LIN {X 0,Y 172.434,Z 372.599,A -85,B 0,C 180,E1 -23622.803,E2 -23622.803} C_VEL
LIN {X 0,Y 167.922,Z 377.389,A -85,B 0,C 180,E1 -23626.32,E2 -23626.32} C_VEL
LIN {X 0,Y 163.411,Z 381.78,A -85,B 0,C 180,E1 -23630.712,E2 -23630.712} C_VEL
LIN {X 0,Y 159.956,Z 384.766,A -85,B 0,C 180,E1 -23635.163,E2 -23635.163} C_VEL
LIN {X 0,Y 157.016,Z 386.825,A -85,B 0,C 180,E1 -23640.5,E2 -23640.5} C_VEL
LIN {X 0,Y 155.23,Z 387.379,A -85,B 0,C 180,E1 -23645.95,E2 -23645.95} C_VEL
LIN {X 0,Y 154.433,Z 386.492,A -85,B 0,C 180,E1 -23651.42,E2 -23651.42} C_VEL
LIN {X 0,Y 154.339,Z 385.518,A -85,B 0,C 180,E1 -23654.141,E2 -23654.141} C_VEL
LIN {X 0,Y 154.579,Z 382.511,A -85,B 0,C 180,E1 -23659.518,E2 -23659.518} C_VEL
LIN {X 0,Y 155.438,Z 378.809,A -85,B 0,C 180,E1 -23664.003,E2 -23664.003} C_VEL
LIN {X 0,Y 156.803,Z 373.593,A -85,B 0,C 180,E1 -23668.712,E2 -23668.712} C_VEL
LIN {X 0,Y 158.828,Z 367.169,A -85,B 0,C 180,E1 -23673.167,E2 -23673.167} C_VEL
LIN {X 0,Y 161.651,Z 359.176,A -85,B 0,C 180,E1 -23677.491,E2 -23677.491} C_VEL
LIN {X 0,Y 164.911,Z 350.124,A -85,B 0,C 180,E1 -23681.341,E2 -23681.341} C_VEL
LIN {X 0,Y 168.005,Z 340.788,A -85,B 0,C 180,E1 -23684.533,E2 -23684.533} C_VEL
LIN {X 0,Y 170.897,Z 331.765,A -85,B 0,C 180,E1 -23687.035,E2 -23687.035} C_VEL
LIN {X 0,Y 174.236,Z 321.032,A -85,B 0,C 180,E1 -23689.434,E2 -23689.434} C_VEL
LIN {X 0,Y 177.782,Z 307.906,A -85,B 0,C 180,E1 -23691.75,E2 -23691.75} C_VEL
LIN {X 0,Y 180.651,Z 295.009,A -85,B 0,C 180,E1 -23693.497,E2 -23693.497} C_VEL
LIN {X 0,Y 183.069,Z 281.077,A -85,B 0,C 180,E1 -23694.9,E2 -23694.9} C_VEL
LIN {X 0,Y 184.747,Z 267.514,A -85,B 0,C 180,E1 -23695.863,E2 -23695.863} C_VEL
LIN {X 0,Y 185.971,Z 252.484,A -85,B 0,C 180,E1 -23696.51,E2 -23696.51} C_VEL
LIN {X 0,Y 189.711,Z 192.551,A -85,B 0,C 180,E1 -23698.519,E2 -23698.519} C_VEL
LIN {X 0,Y 186.693,Z 185.07,A -85,B 0,C 180,E1 -23699.624,E2 -23699.624} C_VEL
LIN {X 0,Y 180.33,Z 172.464,A -85,B 0,C 180,E1 -23701.969,E2 -23701.969} C_VEL
LIN {X 0,Y 173.877,Z 161.345,A -85,B 0,C 180,E1 -23704.503,E2 -23704.503} C_VEL
LIN {X 0,Y 168.485,Z 153.177,A -85,B 0,C 180,E1 -23706.795,E2 -23706.795} C_VEL
LIN {X 0,Y 166.15,Z 149.74,A -85,B 0,C 180,E1 -23707.86,E2 -23707.86} C_VEL
LIN {X 0,Y 163.658,Z 146.027,A -85,B 0,C 180,E1 -23709.057,E2 -23709.057} C_VEL
LIN {X 0,Y 161.372,Z 143.032,A -85,B 0,C 180,E1 -23710.186,E2 -23710.186} C_VEL
LIN {X 0,Y 160.594,Z 141.677,A -85,B 0,C 180,E1 -23710.607,E2 -23710.607} C_VEL
LIN {X 0,Y 158.312,Z 139.434,A -85,B 0,C 180,E1 -23711.764,E2 -23711.764} C_VEL
LIN {X 0,Y 157.313,Z 136.739,A -85,B 0,C 180,E1 -23712.416,E2 -23712.416} C_VEL
LIN {X 0,Y 157.297,Z 136.491,A -85,B 0,C 180,E1 -23712.514,E2 -23712.514} C_VEL
LIN {X 0,Y 157.271,Z 136.517,A -85,B 0,C 180,E1 -23717.922,E2 -23717.922} C_VEL
LIN {X 0,Y 157.301,Z 136.485,A -85,B 0,C 180,E1 -23723.528,E2 -23723.528} C_VEL
LIN {X 0,Y 157.271,Z 136.508,A -85,B 0,C 180,E1 -23728.102,E2 -23728.102} C_VEL
LIN {X 0,Y 157.305,Z 136.482,A -85,B 0,C 180,E1 -23733.473,E2 -23733.473} C_VEL
LIN {X 0,Y 157.429,Z 136.489,A -85,B 0,C 180,E1 -23739.623,E2 -23739.623} C_VEL
LIN {X 0,Y 157.474,Z 136.485,A -85,B 0,C 180,E1 -23744.477,E2 -23744.477} C_VEL
LIN {X 0,Y 157.757,Z 136.45,A -85,B 0,C 180,E1 -23749.744,E2 -23749.744} C_VEL
LIN {X 0,Y 157.809,Z 136.411,A -85,B 0,C 180,E1 -23752.331,E2 -23752.331} C_VEL
LIN {X 0,Y 158.249,Z 136.394,A -85,B 0,C 180,E1 -23760.008,E2 -23760.008} C_VEL
LIN {X 0,Y 157.802,Z 136.438,A -85,B 0,C 180,E1 -23767.686,E2 -23767.686} C_VEL
LIN {X 0,Y 157.678,Z 136.463,A -85,B 0,C 180,E1 -23771.33,E2 -23771.33} C_VEL
LIN {X 0,Y 157.474,Z 136.493,A -85,B 0,C 180,E1 -23775.54,E2 -23775.54} C_VEL
LIN {X 0,Y 157.368,Z 136.504,A -85,B 0,C 180,E1 -23780.941,E2 -23780.941} C_VEL
LIN {X 0,Y 157.314,Z 136.503,A -85,B 0,C 180,E1 -23786.693,E2 -23786.693} C_VEL
LIN {X 0,Y 157.359,Z 136.499,A -85,B 0,C 180,E1 -23791.196,E2 -23791.196} C_VEL
LIN {X 0,Y 158.146,Z 139.101,A -85,B 0,C 180,E1 -23791.771,E2 -23791.771} C_VEL
LIN {X 0,Y 160.016,Z 141.285,A -85,B 0,C 180,E1 -23792.745,E2 -23792.745} C_VEL
LIN {X 0,Y 160.917,Z 142.2,A -85,B 0,C 180,E1 -23793.19,E2 -23793.19} C_VEL
LIN {X 0,Y 163.097,Z 145.539,A -85,B 0,C 180,E1 -23794.306,E2 -23794.306} C_VEL
LIN {X 0,Y 164.461,Z 147.244,A -85,B 0,C 180,E1 -23794.953,E2 -23794.953} C_VEL
LIN {X 0,Y 171.828,Z 158.11,A -85,B 0,C 180,E1 -23798.265,E2 -23798.265} C_VEL
LIN {X 0,Y 175.525,Z 165.073,A -85,B 0,C 180,E1 -23799.847,E2 -23799.847} C_VEL
LIN {X 0,Y 181.579,Z 178.258,A -85,B 0,C 180,E1 -23802.315,E2 -23802.315} C_VEL
LIN {X 0,Y 186.446,Z 190.92,A -85,B 0,C 180,E1 -23804.231,E2 -23804.231} C_VEL
LIN {X 0,Y 189.413,Z 199.801,A -85,B 0,C 180,E1 -23805.386,E2 -23805.386} C_VEL
LIN {X 0,Y 185.075,Z 271.299,A -85,B 0,C 180,E1 -23807.901,E2 -23807.901} C_VEL
LIN {X 0,Y 183.311,Z 285.784,A -85,B 0,C 180,E1 -23808.784,E2 -23808.784} C_VEL
LIN {X 0,Y 180.955,Z 299.227,A -85,B 0,C 180,E1 -23809.982,E2 -23809.982} C_VEL
LIN {X 0,Y 178.058,Z 312.27,A -85,B 0,C 180,E1 -23811.567,E2 -23811.567} C_VEL
LIN {X 0,Y 174.864,Z 324.428,A -85,B 0,C 180,E1 -23813.507,E2 -23813.507} C_VEL
LIN {X 0,Y 174.269,Z 326.771,A -85,B 0,C 180,E1 -23813.944,E2 -23813.944} C_VEL
LIN {X 0,Y 172.717,Z 330.07,A -85,B 0,C 180,E1 -23814.493,E2 -23814.493} C_VEL
LIN {X 0,Y 164.418,Z 340.003,A -85,B 0,C 180,E1 -23815.867,E2 -23815.867} C_VEL
LIN {X 0,Y 162.874,Z 343.02,A -85,B 0,C 180,E1 -23816.573,E2 -23816.573} C_VEL
LIN {X 0,Y 159.287,Z 352.662,A -85,B 0,C 180,E1 -23819.514,E2 -23819.514} C_VEL
LIN {X 0,Y 155.811,Z 362.205,A -85,B 0,C 180,E1 -23823.193,E2 -23823.193} C_VEL
LIN {X 0,Y 152.861,Z 370.256,A -85,B 0,C 180,E1 -23827.093,E2 -23827.093} C_VEL
LIN {X 0,Y 150.785,Z 376.646,A -85,B 0,C 180,E1 -23830.962,E2 -23830.962} C_VEL
LIN {X 0,Y 149.126,Z 382.032,A -85,B 0,C 180,E1 -23834.981,E2 -23834.981} C_VEL
LIN {X 0,Y 148.16,Z 386.429,A -85,B 0,C 180,E1 -23839.066,E2 -23839.066} C_VEL
LIN {X 0,Y 147.695,Z 389.897,A -85,B 0,C 180,E1 -23843.172,E2 -23843.172} C_VEL
LIN {X 0,Y 147.649,Z 393.153,A -85,B 0,C 180,E1 -23848.614,E2 -23848.614} C_VEL
LIN {X 0,Y 147.627,Z 394.629,A -85,B 0,C 180,E1 -23852.733,E2 -23852.733} C_VEL
LIN {X 0,Y 147.843,Z 395.435,A -85,B 0,C 180,E1 -23858.203,E2 -23858.203} C_VEL
LIN {X 0,Y 148.985,Z 394.938,A -85,B 0,C 180,E1 -23863.646,E2 -23863.646} C_VEL
LIN {X 0,Y 151.32,Z 393.151,A -85,B 0,C 180,E1 -23868.976,E2 -23868.976} C_VEL
LIN {X 0,Y 154.924,Z 390.039,A -85,B 0,C 180,E1 -23874.101,E2 -23874.101} C_VEL
LIN {X 0,Y 159.574,Z 385.523,A -85,B 0,C 180,E1 -23878.981,E2 -23878.981} C_VEL
LIN {X 0,Y 163.865,Z 381.086,A -85,B 0,C 180,E1 -23882.423,E2 -23882.423} C_VEL
LIN {X 0,Y 169.627,Z 374.725,A -85,B 0,C 180,E1 -23886.19,E2 -23886.19} C_VEL
LIN {X 0,Y 176.159,Z 366.857,A -85,B 0,C 180,E1 -23889.671,E2 -23889.671} C_VEL
LIN {X 0,Y 182.278,Z 358.665,A -85,B 0,C 180,E1 -23892.438,E2 -23892.438} C_VEL
LIN {X 0,Y 187.822,Z 350.229,A -85,B 0,C 180,E1 -23894.726,E2 -23894.726} C_VEL
LIN {X 0,Y 194.472,Z 339.024,A -85,B 0,C 180,E1 -23897.042,E2 -23897.042} C_VEL
LIN {X 0,Y 200.429,Z 327.209,A -85,B 0,C 180,E1 -23898.933,E2 -23898.933} C_VEL
LIN {X 0,Y 205.426,Z 315.612,A -85,B 0,C 180,E1 -23900.337,E2 -23900.337} C_VEL
LIN {X 0,Y 210.231,Z 302.016,A -85,B 0,C 180,E1 -23901.587,E2 -23901.587} C_VEL
LIN {X 0,Y 214.074,Z 287.872,A -85,B 0,C 180,E1 -23902.515,E2 -23902.515} C_VEL
LIN {X 0,Y 216.731,Z 274.058,A -85,B 0,C 180,E1 -23903.154,E2 -23903.154} C_VEL
LIN {X 0,Y 218.512,Z 258.395,A -85,B 0,C 180,E1 -23903.633,E2 -23903.633} C_VEL
LIN {X 0,Y 220.891,Z 229.848,A -85,B 0,C 180,E1 -23904.433,E2 -23904.433} C_VEL
LIN {X 0,Y 216.996,Z 220.369,A -85,B 0,C 180,E1 -23907.047,E2 -23907.047} C_VEL
LIN {X 0,Y 213.245,Z 212.121,A -85,B 0,C 180,E1 -23909.877,E2 -23909.877} C_VEL
LIN {X 0,Y 209.714,Z 204.899,A -85,B 0,C 180,E1 -23912.975,E2 -23912.975} C_VEL
LIN {X 0,Y 207.676,Z 201.073,A -85,B 0,C 180,E1 -23915.013,E2 -23915.013} C_VEL
LIN {X 0,Y 205.063,Z 196.287,A -85,B 0,C 180,E1 -23918.072,E2 -23918.072} C_VEL
LIN {X 0,Y 202.418,Z 191.695,A -85,B 0,C 180,E1 -23922.156,E2 -23922.156} C_VEL
LIN {X 0,Y 199.839,Z 187.624,A -85,B 0,C 180,E1 -23930.122,E2 -23930.122} C_VEL
LIN {X 0,Y 199.808,Z 186.636,A -85,B 0,C 180,E1 -23931.906,E2 -23931.906} C_VEL
LIN {X 0,Y 199.886,Z 187.122,A -85,B 0,C 180,E1 -23934.206,E2 -23934.206} C_VEL
LIN {X 0,Y 200.605,Z 188.988,A -85,B 0,C 180,E1 -23937.986,E2 -23937.986} C_VEL
LIN {X 0,Y 202.823,Z 192.052,A -85,B 0,C 180,E1 -23942.94,E2 -23942.94} C_VEL
LIN {X 0,Y 205.027,Z 195.594,A -85,B 0,C 180,E1 -23946.218,E2 -23946.218} C_VEL
LIN {X 0,Y 208.548,Z 201.132,A -85,B 0,C 180,E1 -23950.141,E2 -23950.141} C_VEL
LIN {X 0,Y 211.159,Z 205.435,A -85,B 0,C 180,E1 -23952.548,E2 -23952.548} C_VEL
LIN {X 0,Y 214.843,Z 211.525,A -85,B 0,C 180,E1 -23955.474,E2 -23955.474} C_VEL
LIN {X 0,Y 218.814,Z 218.863,A -85,B 0,C 180,E1 -23958.211,E2 -23958.211} C_VEL
LIN {X 0,Y 221.356,Z 224.64,A -85,B 0,C 180,E1 -23959.855,E2 -23959.855} C_VEL
LIN {X 0,Y 217.702,Z 264.642,A -85,B 0,C 180,E1 -23960.966,E2 -23960.966} C_VEL
LIN {X 0,Y 215.161,Z 279.353,A -85,B 0,C 180,E1 -23961.629,E2 -23961.629} C_VEL
LIN {X 0,Y 211.978,Z 292.142,A -85,B 0,C 180,E1 -23962.449,E2 -23962.449} C_VEL
LIN {X 0,Y 208.023,Z 304.769,A -85,B 0,C 180,E1 -23963.587,E2 -23963.587} C_VEL
LIN {X 0,Y 203.226,Z 317.121,A -85,B 0,C 180,E1 -23965.045,E2 -23965.045} C_VEL
LIN {X 0,Y 197.798,Z 328.646,A -85,B 0,C 180,E1 -23966.777,E2 -23966.777} C_VEL
LIN {X 0,Y 191.693,Z 339.69,A -85,B 0,C 180,E1 -23968.911,E2 -23968.911} C_VEL
LIN {X 0,Y 185.342,Z 349.716,A -85,B 0,C 180,E1 -23971.435,E2 -23971.435} C_VEL
LIN {X 0,Y 178.81,Z 358.726,A -85,B 0,C 180,E1 -23974.367,E2 -23974.367} C_VEL
LIN {X 0,Y 172.596,Z 366.369,A -85,B 0,C 180,E1 -23977.635,E2 -23977.635} C_VEL
LIN {X 0,Y 167.363,Z 372.189,A -85,B 0,C 180,E1 -23980.894,E2 -23980.894} C_VEL
LIN {X 0,Y 162.509,Z 377.101,A -85,B 0,C 180,E1 -23984.469,E2 -23984.469} C_VEL
LIN {X 0,Y 158.316,Z 380.997,A -85,B 0,C 180,E1 -23988.245,E2 -23988.245} C_VEL
LIN {X 0,Y 153.78,Z 384.714,A -85,B 0,C 180,E1 -23993.546,E2 -23993.546} C_VEL
LIN {X 0,Y 150.481,Z 386.891,A -85,B 0,C 180,E1 -23999.083,E2 -23999.083} C_VEL
LIN {X 0,Y 148.417,Z 387.597,A -85,B 0,C 180,E1 -24004.771,E2 -24004.771} C_VEL
LIN {X 0,Y 147.399,Z 386.836,A -85,B 0,C 180,E1 -24010.499,E2 -24010.499} C_VEL
LIN {X 0,Y 147.257,Z 385.916,A -85,B 0,C 180,E1 -24013.356,E2 -24013.356} C_VEL
LIN {X 0,Y 147.419,Z 383.018,A -85,B 0,C 180,E1 -24019.003,E2 -24019.003} C_VEL
LIN {X 0,Y 148.342,Z 379.058,A -85,B 0,C 180,E1 -24024.114,E2 -24024.114} C_VEL
LIN {X 0,Y 149.634,Z 374.336,A -85,B 0,C 180,E1 -24028.651,E2 -24028.651} C_VEL
LIN {X 0,Y 151.656,Z 368.049,A -85,B 0,C 180,E1 -24033.317,E2 -24033.317} C_VEL
LIN {X 0,Y 154.593,Z 360.199,A -85,B 0,C 180,E1 -24037.835,E2 -24037.835} C_VEL
LIN {X 0,Y 158.013,Z 351.07,A -85,B 0,C 180,E1 -24041.952,E2 -24041.952} C_VEL
LIN {X 0,Y 161.157,Z 342.173,A -85,B 0,C 180,E1 -24045.165,E2 -24045.165} C_VEL
LIN {X 0,Y 164.461,Z 332.322,A -85,B 0,C 180,E1 -24048.044,E2 -24048.044} C_VEL
LIN {X 0,Y 167.934,Z 321.663,A -85,B 0,C 180,E1 -24050.514,E2 -24050.514} C_VEL
LIN {X 0,Y 171.179,Z 310.228,A -85,B 0,C 180,E1 -24052.634,E2 -24052.634} C_VEL
LIN {X 0,Y 174.173,Z 297.857,A -85,B 0,C 180,E1 -24054.427,E2 -24054.427} C_VEL
LIN {X 0,Y 176.78,Z 284.203,A -85,B 0,C 180,E1 -24055.929,E2 -24055.929} C_VEL
LIN {X 0,Y 178.701,Z 270.115,A -85,B 0,C 180,E1 -24057.044,E2 -24057.044} C_VEL
LIN {X 0,Y 180.021,Z 256.632,A -85,B 0,C 180,E1 -24057.695,E2 -24057.695} C_VEL
LIN {X 0,Y 184.017,Z 194.279,A -85,B 0,C 180,E1 -24059.843,E2 -24059.843} C_VEL
LIN {X 0,Y 180.637,Z 186.301,A -85,B 0,C 180,E1 -24061.153,E2 -24061.153} C_VEL
LIN {X 0,Y 173.704,Z 172.894,A -85,B 0,C 180,E1 -24063.898,E2 -24063.898} C_VEL
LIN {X 0,Y 165.781,Z 159.766,A -85,B 0,C 180,E1 -24067.36,E2 -24067.36} C_VEL
LIN {X 0,Y 159.846,Z 151.212,A -85,B 0,C 180,E1 -24070.261,E2 -24070.261} C_VEL
LIN {X 0,Y 157.001,Z 147.249,A -85,B 0,C 180,E1 -24071.787,E2 -24071.787} C_VEL
LIN {X 0,Y 154.581,Z 144.195,A -85,B 0,C 180,E1 -24073.144,E2 -24073.144} C_VEL
LIN {X 0,Y 153.612,Z 142.541,A -85,B 0,C 180,E1 -24073.741,E2 -24073.741} C_VEL
LIN {X 0,Y 151.409,Z 140.485,A -85,B 0,C 180,E1 -24075.023,E2 -24075.023} C_VEL
LIN {X 0,Y 150.337,Z 137.963,A -85,B 0,C 180,E1 -24075.8,E2 -24075.8} C_VEL
LIN {X 0,Y 150.25,Z 137.377,A -85,B 0,C 180,E1 -24075.974,E2 -24075.974} C_VEL
LIN {X 0,Y 150.213,Z 137.38,A -85,B 0,C 180,E1 -24079.093,E2 -24079.093} C_VEL
LIN {X 0,Y 150.215,Z 137.36,A -85,B 0,C 180,E1 -24082.683,E2 -24082.683} C_VEL
LIN {X 0,Y 150.195,Z 137.395,A -85,B 0,C 180,E1 -24087.372,E2 -24087.372} C_VEL
LIN {X 0,Y 150.225,Z 137.355,A -85,B 0,C 180,E1 -24092.724,E2 -24092.724} C_VEL
LIN {X 0,Y 150.372,Z 137.369,A -85,B 0,C 180,E1 -24099.176,E2 -24099.176} C_VEL
LIN {X 0,Y 150.382,Z 137.372,A -85,B 0,C 180,E1 -24103.725,E2 -24103.725} C_VEL
LIN {X 0,Y 150.674,Z 137.335,A -85,B 0,C 180,E1 -24109.256,E2 -24109.256} C_VEL
LIN {X 0,Y 150.748,Z 137.292,A -85,B 0,C 180,E1 -24111.969,E2 -24111.969} C_VEL
LIN {X 0,Y 151.21,Z 137.271,A -85,B 0,C 180,E1 -24120.009,E2 -24120.009} C_VEL
LIN {X 0,Y 150.738,Z 137.321,A -85,B 0,C 180,E1 -24128.049,E2 -24128.049} C_VEL
LIN {X 0,Y 150.609,Z 137.342,A -85,B 0,C 180,E1 -24131.516,E2 -24131.516} C_VEL
LIN {X 0,Y 150.378,Z 137.372,A -85,B 0,C 180,E1 -24136.293,E2 -24136.293} C_VEL
LIN {X 0,Y 150.349,Z 137.379,A -85,B 0,C 180,E1 -24140.801,E2 -24140.801} C_VEL
LIN {X 0,Y 150.242,Z 137.379,A -85,B 0,C 180,E1 -24147.46,E2 -24147.46} C_VEL
LIN {X 0,Y 150.237,Z 137.471,A -85,B 0,C 180,E1 -24147.735,E2 -24147.735} C_VEL
LIN {X 0,Y 151.071,Z 140.001,A -85,B 0,C 180,E1 -24148.393,E2 -24148.393} C_VEL
LIN {X 0,Y 153.047,Z 142.213,A -85,B 0,C 180,E1 -24149.589,E2 -24149.589} C_VEL
LIN {X 0,Y 154.115,Z 143.128,A -85,B 0,C 180,E1 -24150.187,E2 -24150.187} C_VEL
LIN {X 0,Y 155.933,Z 146.168,A -85,B 0,C 180,E1 -24151.28,E2 -24151.28} C_VEL
LIN {X 0,Y 157.726,Z 148.199,A -85,B 0,C 180,E1 -24152.239,E2 -24152.239} C_VEL
LIN {X 0,Y 161.837,Z 154.17,A -85,B 0,C 180,E1 -24154.379,E2 -24154.379} C_VEL
LIN {X 0,Y 166.797,Z 161.553,A -85,B 0,C 180,E1 -24156.738,E2 -24156.738} C_VEL
LIN {X 0,Y 170.002,Z 167.123,A -85,B 0,C 180,E1 -24158.189,E2 -24158.189} C_VEL
LIN {X 0,Y 175.768,Z 179.62,A -85,B 0,C 180,E1 -24160.731,E2 -24160.731} C_VEL
LIN {X 0,Y 180.106,Z 190.708,A -85,B 0,C 180,E1 -24162.565,E2 -24162.565} C_VEL
LIN {X 0,Y 183.751,Z 201.211,A -85,B 0,C 180,E1 -24164.065,E2 -24164.065} C_VEL
LIN {X 0,Y 179.412,Z 270.362,A -85,B 0,C 180,E1 -24166.536,E2 -24166.536} C_VEL
LIN {X 0,Y 177.609,Z 285.111,A -85,B 0,C 180,E1 -24167.442,E2 -24167.442} C_VEL
LIN {X 0,Y 175.335,Z 298.041,A -85,B 0,C 180,E1 -24168.6,E2 -24168.6} C_VEL
LIN {X 0,Y 172.549,Z 310.475,A -85,B 0,C 180,E1 -24170.1,E2 -24170.1} C_VEL
LIN {X 0,Y 169.567,Z 321.592,A -85,B 0,C 180,E1 -24171.822,E2 -24171.822} C_VEL
LIN {X 0,Y 165.79,Z 334.145,A -85,B 0,C 180,E1 -24174.351,E2 -24174.351} C_VEL
LIN {X 0,Y 163.142,Z 342.089,A -85,B 0,C 180,E1 -24176.318,E2 -24176.318} C_VEL
LIN {X 0,Y 162.874,Z 343.02,A -85,B 0,C 180,E1 -24176.573,E2 -24176.573} C_VEL
LIN {X 0,Y 161.674,Z 346.003,A -85,B 0,C 180,E1 -24177.372,E2 -24177.372} C_VEL
LIN {X 0,Y 158.954,Z 350.251,A -85,B 0,C 180,E1 -24178.484,E2 -24178.484} C_VEL
LIN {X 0,Y 151.328,Z 359.278,A -85,B 0,C 180,E1 -24181.218,E2 -24181.218} C_VEL
LIN {X 0,Y 148.863,Z 362.997,A -85,B 0,C 180,E1 -24182.715,E2 -24182.715} C_VEL
LIN {X 0,Y 148.325,Z 364.196,A -85,B 0,C 180,E1 -24183.278,E2 -24183.278} C_VEL
LIN {X 0,Y 145.48,Z 371.68,A -85,B 0,C 180,E1 -24187.269,E2 -24187.269} C_VEL
LIN {X 0,Y 143.375,Z 377.942,A -85,B 0,C 180,E1 -24191.425,E2 -24191.425} C_VEL
LIN {X 0,Y 141.788,Z 383.097,A -85,B 0,C 180,E1 -24195.655,E2 -24195.655} C_VEL
LIN {X 0,Y 140.777,Z 388.386,A -85,B 0,C 180,E1 -24201.391,E2 -24201.391} C_VEL
LIN {X 0,Y 140.522,Z 392.095,A -85,B 0,C 180,E1 -24207.137,E2 -24207.137} C_VEL
LIN {X 0,Y 140.588,Z 393.663,A -85,B 0,C 180,E1 -24210.691,E2 -24210.691} C_VEL
LIN {X 0,Y 140.563,Z 394.946,A -85,B 0,C 180,E1 -24215.743,E2 -24215.743} C_VEL
LIN {X 0,Y 141.31,Z 395.169,A -85,B 0,C 180,E1 -24221.479,E2 -24221.479} C_VEL
LIN {X 0,Y 143.105,Z 394.102,A -85,B 0,C 180,E1 -24227.141,E2 -24227.141} C_VEL
LIN {X 0,Y 146.34,Z 391.74,A -85,B 0,C 180,E1 -24232.598,E2 -24232.598} C_VEL
LIN {X 0,Y 150.736,Z 388.022,A -85,B 0,C 180,E1 -24237.795,E2 -24237.795} C_VEL
LIN {X 0,Y 156.307,Z 382.845,A -85,B 0,C 180,E1 -24242.657,E2 -24242.657} C_VEL
LIN {X 0,Y 161.251,Z 377.865,A -85,B 0,C 180,E1 -24246.047,E2 -24246.047} C_VEL
LIN {X 0,Y 167.733,Z 370.778,A -85,B 0,C 180,E1 -24249.72,E2 -24249.72} C_VEL
LIN {X 0,Y 174.979,Z 362.045,A -85,B 0,C 180,E1 -24253.067,E2 -24253.067} C_VEL
LIN {X 0,Y 181.647,Z 352.677,A -85,B 0,C 180,E1 -24255.851,E2 -24255.851} C_VEL
LIN {X 0,Y 188.537,Z 341.955,A -85,B 0,C 180,E1 -24258.209,E2 -24258.209} C_VEL
LIN {X 0,Y 194.676,Z 330.775,A -85,B 0,C 180,E1 -24260.103,E2 -24260.103} C_VEL
LIN {X 0,Y 199.711,Z 320.021,A -85,B 0,C 180,E1 -24261.54,E2 -24261.54} C_VEL
LIN {X 0,Y 204.977,Z 306.632,A -85,B 0,C 180,E1 -24262.865,E2 -24262.865} C_VEL
LIN {X 0,Y 208.983,Z 293.745,A -85,B 0,C 180,E1 -24263.818,E2 -24263.818} C_VEL
LIN {X 0,Y 212.248,Z 279.853,A -85,B 0,C 180,E1 -24264.54,E2 -24264.54} C_VEL
LIN {X 0,Y 214.303,Z 265.982,A -85,B 0,C 180,E1 -24265.075,E2 -24265.075} C_VEL
LIN {X 0,Y 217.278,Z 233.024,A -85,B 0,C 180,E1 -24265.975,E2 -24265.975} C_VEL
LIN {X 0,Y 213.936,Z 224.705,A -85,B 0,C 180,E1 -24268.406,E2 -24268.406} C_VEL
LIN {X 0,Y 210.605,Z 216.971,A -85,B 0,C 180,E1 -24271.177,E2 -24271.177} C_VEL
LIN {X 0,Y 207.632,Z 210.653,A -85,B 0,C 180,E1 -24273.999,E2 -24273.999} C_VEL
LIN {X 0,Y 206,Z 207.434,A -85,B 0,C 180,E1 -24275.748,E2 -24275.748} C_VEL
LIN {X 0,Y 203.52,Z 202.66,A -85,B 0,C 180,E1 -24278.852,E2 -24278.852} C_VEL
LIN {X 0,Y 201.072,Z 198.429,A -85,B 0,C 180,E1 -24282.95,E2 -24282.95} C_VEL
LIN {X 0,Y 198.91,Z 194.245,A -85,B 0,C 180,E1 -24290.965,E2 -24290.965} C_VEL
LIN {X 0,Y 198.924,Z 193.683,A -85,B 0,C 180,E1 -24291.869,E2 -24291.869} C_VEL
LIN {X 0,Y 198.996,Z 194.179,A -85,B 0,C 180,E1 -24294.18,E2 -24294.18} C_VEL
LIN {X 0,Y 199.705,Z 196.1,A -85,B 0,C 180,E1 -24297.977,E2 -24297.977} C_VEL
LIN {X 0,Y 201.661,Z 198.942,A -85,B 0,C 180,E1 -24302.52,E2 -24302.52} C_VEL
LIN {X 0,Y 203.754,Z 202.399,A -85,B 0,C 180,E1 -24305.795,E2 -24305.795} C_VEL
LIN {X 0,Y 206.926,Z 207.677,A -85,B 0,C 180,E1 -24309.511,E2 -24309.511} C_VEL
LIN {X 0,Y 209.409,Z 211.936,A -85,B 0,C 180,E1 -24311.917,E2 -24311.917} C_VEL
LIN {X 0,Y 212.817,Z 217.808,A -85,B 0,C 180,E1 -24314.761,E2 -24314.761} C_VEL
LIN {X 0,Y 216.299,Z 224.569,A -85,B 0,C 180,E1 -24317.317,E2 -24317.317} C_VEL
LIN {X 0,Y 217.698,Z 227.796,A -85,B 0,C 180,E1 -24318.285,E2 -24318.285} C_VEL
LIN {X 0,Y 214.216,Z 264.881,A -85,B 0,C 180,E1 -24319.325,E2 -24319.325} C_VEL
LIN {X 0,Y 211.68,Z 279.215,A -85,B 0,C 180,E1 -24319.958,E2 -24319.958} C_VEL
LIN {X 0,Y 208.198,Z 292.836,A -85,B 0,C 180,E1 -24320.825,E2 -24320.825} C_VEL
LIN {X 0,Y 203.74,Z 306.414,A -85,B 0,C 180,E1 -24322.059,E2 -24322.059} C_VEL
LIN {X 0,Y 198.461,Z 319.232,A -85,B 0,C 180,E1 -24323.603,E2 -24323.603} C_VEL
LIN {X 0,Y 192.644,Z 330.836,A -85,B 0,C 180,E1 -24325.401,E2 -24325.401} C_VEL
LIN {X 0,Y 186.307,Z 341.587,A -85,B 0,C 180,E1 -24327.56,E2 -24327.56} C_VEL
LIN {X 0,Y 179.179,Z 352.073,A -85,B 0,C 180,E1 -24330.349,E2 -24330.349} C_VEL
LIN {X 0,Y 172.474,Z 360.68,A -85,B 0,C 180,E1 -24333.344,E2 -24333.344} C_VEL
LIN {X 0,Y 165.318,Z 368.825,A -85,B 0,C 180,E1 -24337.141,E2 -24337.141} C_VEL
LIN {X 0,Y 158.328,Z 375.895,A -85,B 0,C 180,E1 -24341.733,E2 -24341.733} C_VEL
LIN {X 0,Y 152.72,Z 380.836,A -85,B 0,C 180,E1 -24346.343,E2 -24346.343} C_VEL
LIN {X 0,Y 147.75,Z 384.671,A -85,B 0,C 180,E1 -24351.798,E2 -24351.798} C_VEL
LIN {X 0,Y 144.038,Z 386.959,A -85,B 0,C 180,E1 -24357.535,E2 -24357.535} C_VEL
LIN {X 0,Y 141.645,Z 387.776,A -85,B 0,C 180,E1 -24363.473,E2 -24363.473} C_VEL
LIN {X 0,Y 140.387,Z 387.16,A -85,B 0,C 180,E1 -24369.482,E2 -24369.482} C_VEL
LIN {X 0,Y 140.178,Z 386.311,A -85,B 0,C 180,E1 -24372.489,E2 -24372.489} C_VEL
LIN {X 0,Y 140.118,Z 385.099,A -85,B 0,C 180,E1 -24375.472,E2 -24375.472} C_VEL
LIN {X 0,Y 140.688,Z 381.582,A -85,B 0,C 180,E1 -24381.377,E2 -24381.377} C_VEL
LIN {X 0,Y 141.633,Z 377.992,A -85,B 0,C 180,E1 -24385.727,E2 -24385.727} C_VEL
LIN {X 0,Y 142.961,Z 373.442,A -85,B 0,C 180,E1 -24389.996,E2 -24389.996} C_VEL
LIN {X 0,Y 145.315,Z 366.88,A -85,B 0,C 180,E1 -24394.851,E2 -24394.851} C_VEL
LIN {X 0,Y 148.49,Z 358.741,A -85,B 0,C 180,E1 -24399.531,E2 -24399.531} C_VEL
LIN {X 0,Y 151.856,Z 350.216,A -85,B 0,C 180,E1 -24403.376,E2 -24403.376} C_VEL
LIN {X 0,Y 154.934,Z 341.78,A -85,B 0,C 180,E1 -24406.466,E2 -24406.466} C_VEL
LIN {X 0,Y 158.099,Z 332.875,A -85,B 0,C 180,E1 -24409.134,E2 -24409.134} C_VEL
LIN {X 0,Y 161.697,Z 322.294,A -85,B 0,C 180,E1 -24411.677,E2 -24411.677} C_VEL
LIN {X 0,Y 165.521,Z 309.361,A -85,B 0,C 180,E1 -24414.118,E2 -24414.118} C_VEL
LIN {X 0,Y 168.854,Z 295.733,A -85,B 0,C 180,E1 -24416.076,E2 -24416.076} C_VEL
LIN {X 0,Y 171.364,Z 282.654,A -85,B 0,C 180,E1 -24417.473,E2 -24417.473} C_VEL
LIN {X 0,Y 173.291,Z 268.647,A -85,B 0,C 180,E1 -24418.538,E2 -24418.538} C_VEL
LIN {X 0,Y 174.654,Z 253.784,A -85,B 0,C 180,E1 -24419.209,E2 -24419.209} C_VEL
LIN {X 0,Y 178.527,Z 196.37,A -85,B 0,C 180,E1 -24421.201,E2 -24421.201} C_VEL
LIN {X 0,Y 173.66,Z 185.677,A -85,B 0,C 180,E1 -24423.19,E2 -24423.19} C_VEL
LIN {X 0,Y 167.451,Z 174.03,A -85,B 0,C 180,E1 -24425.879,E2 -24425.879} C_VEL
LIN {X 0,Y 161.402,Z 164.096,A -85,B 0,C 180,E1 -24428.749,E2 -24428.749} C_VEL
LIN {X 0,Y 156.292,Z 156.503,A -85,B 0,C 180,E1 -24431.433,E2 -24431.433} C_VEL
LIN {X 0,Y 153.741,Z 152.93,A -85,B 0,C 180,E1 -24432.883,E2 -24432.883} C_VEL
LIN {X 0,Y 151.142,Z 149.338,A -85,B 0,C 180,E1 -24434.449,E2 -24434.449} C_VEL
LIN {X 0,Y 149.668,Z 147.686,A -85,B 0,C 180,E1 -24435.355,E2 -24435.355} C_VEL
LIN {X 0,Y 147.635,Z 144.821,A -85,B 0,C 180,E1 -24436.716,E2 -24436.716} C_VEL
LIN {X 0,Y 147.11,Z 143.766,A -85,B 0,C 180,E1 -24437.11,E2 -24437.11} C_VEL
LIN {X 0,Y 144.647,Z 141.795,A -85,B 0,C 180,E1 -24438.772,E2 -24438.772} C_VEL
LIN {X 0,Y 143.355,Z 139.317,A -85,B 0,C 180,E1 -24439.839,E2 -24439.839} C_VEL
LIN {X 0,Y 143.108,Z 138.249,A -85,B 0,C 180,E1 -24440.173,E2 -24440.173} C_VEL
LIN {X 0,Y 143.146,Z 138.277,A -85,B 0,C 180,E1 -24446.571,E2 -24446.571} C_VEL
LIN {X 0,Y 143.17,Z 138.229,A -85,B 0,C 180,E1 -24452.07,E2 -24452.07} C_VEL
LIN {X 0,Y 143.293,Z 138.252,A -85,B 0,C 180,E1 -24458.718,E2 -24458.718} C_VEL
LIN {X 0,Y 143.32,Z 138.257,A -85,B 0,C 180,E1 -24462.899,E2 -24462.899} C_VEL
LIN {X 0,Y 143.588,Z 138.222,A -85,B 0,C 180,E1 -24468.719,E2 -24468.719} C_VEL
LIN {X 0,Y 143.669,Z 138.176,A -85,B 0,C 180,E1 -24471.571,E2 -24471.571} C_VEL
LIN {X 0,Y 144.168,Z 138.148,A -85,B 0,C 180,E1 -24480.009,E2 -24480.009} C_VEL
LIN {X 0,Y 143.659,Z 138.206,A -85,B 0,C 180,E1 -24488.448,E2 -24488.448} C_VEL
LIN {X 0,Y 143.543,Z 138.221,A -85,B 0,C 180,E1 -24491.722,E2 -24491.722} C_VEL
LIN {X 0,Y 143.313,Z 138.249,A -85,B 0,C 180,E1 -24497.121,E2 -24497.121} C_VEL
LIN {X 0,Y 143.275,Z 138.26,A -85,B 0,C 180,E1 -24501.264,E2 -24501.264} C_VEL
LIN {X 0,Y 143.165,Z 138.273,A -85,B 0,C 180,E1 -24503.516,E2 -24503.516} C_VEL
LIN {X 0,Y 144.064,Z 140.956,A -85,B 0,C 180,E1 -24504.411,E2 -24504.411} C_VEL
LIN {X 0,Y 146.267,Z 143.299,A -85,B 0,C 180,E1 -24505.981,E2 -24505.981} C_VEL
LIN {X 0,Y 147.298,Z 144.141,A -85,B 0,C 180,E1 -24506.656,E2 -24506.656} C_VEL
LIN {X 0,Y 149.348,Z 147.426,A -85,B 0,C 180,E1 -24508.081,E2 -24508.081} C_VEL
LIN {X 0,Y 151.206,Z 149.365,A -85,B 0,C 180,E1 -24509.221,E2 -24509.221} C_VEL
LIN {X 0,Y 153.756,Z 152.947,A -85,B 0,C 180,E1 -24510.764,E2 -24510.764} C_VEL
LIN {X 0,Y 158.238,Z 159.418,A -85,B 0,C 180,E1 -24513.255,E2 -24513.255} C_VEL
LIN {X 0,Y 164.479,Z 169.07,A -85,B 0,C 180,E1 -24516.369,E2 -24516.369} C_VEL
LIN {X 0,Y 169.701,Z 180.156,A -85,B 0,C 180,E1 -24518.863,E2 -24518.863} C_VEL
LIN {X 0,Y 174.664,Z 192.717,A -85,B 0,C 180,E1 -24521.128,E2 -24521.128} C_VEL
LIN {X 0,Y 178.215,Z 203.213,A -85,B 0,C 180,E1 -24522.706,E2 -24522.706} C_VEL
LIN {X 0,Y 173.76,Z 270.612,A -85,B 0,C 180,E1 -24525.152,E2 -24525.152} C_VEL
LIN {X 0,Y 171.886,Z 285.208,A -85,B 0,C 180,E1 -24526.073,E2 -24526.073} C_VEL
LIN {X 0,Y 169.529,Z 298.064,A -85,B 0,C 180,E1 -24527.252,E2 -24527.252} C_VEL
LIN {X 0,Y 166.638,Z 310.451,A -85,B 0,C 180,E1 -24528.782,E2 -24528.782} C_VEL
LIN {X 0,Y 163.853,Z 320.407,A -85,B 0,C 180,E1 -24530.334,E2 -24530.334} C_VEL
LIN {X 0,Y 160.072,Z 332.884,A -85,B 0,C 180,E1 -24532.87,E2 -24532.87} C_VEL
LIN {X 0,Y 157.556,Z 339.813,A -85,B 0,C 180,E1 -24534.562,E2 -24534.562} C_VEL
LIN {X 0,Y 154.594,Z 348.022,A -85,B 0,C 180,E1 -24536.944,E2 -24536.944} C_VEL
LIN {X 0,Y 150.576,Z 358.308,A -85,B 0,C 180,E1 -24540.659,E2 -24540.659} C_VEL
LIN {X 0,Y 148.325,Z 364.196,A -85,B 0,C 180,E1 -24543.278,E2 -24543.278} C_VEL
LIN {X 0,Y 146.394,Z 367.717,A -85,B 0,C 180,E1 -24544.967,E2 -24544.967} C_VEL
LIN {X 0,Y 141.67,Z 372.978,A -85,B 0,C 180,E1 -24547.735,E2 -24547.735} C_VEL
LIN {X 0,Y 137.134,Z 377.716,A -85,B 0,C 180,E1 -24550.814,E2 -24550.814} C_VEL
LIN {X 0,Y 135.56,Z 380.342,A -85,B 0,C 180,E1 -24552.938,E2 -24552.938} C_VEL
LIN {X 0,Y 134.171,Z 385.462,A -85,B 0,C 180,E1 -24557.91,E2 -24557.91} C_VEL
LIN {X 0,Y 133.588,Z 389.02,A -85,B 0,C 180,E1 -24562.447,E2 -24562.447} C_VEL
LIN {X 0,Y 133.424,Z 391.733,A -85,B 0,C 180,E1 -24566.985,E2 -24566.985} C_VEL
LIN {X 0,Y 133.55,Z 393.076,A -85,B 0,C 180,E1 -24570.004,E2 -24570.004} C_VEL
LIN {X 0,Y 133.475,Z 394.055,A -85,B 0,C 180,E1 -24573.023,E2 -24573.023} C_VEL
LIN {X 0,Y 133.756,Z 395.004,A -85,B 0,C 180,E1 -24579.074,E2 -24579.074} C_VEL
LIN {X 0,Y 135.149,Z 394.656,A -85,B 0,C 180,E1 -24585.075,E2 -24585.075} C_VEL
LIN {X 0,Y 137.905,Z 393.024,A -85,B 0,C 180,E1 -24590.904,E2 -24590.904} C_VEL
LIN {X 0,Y 141.997,Z 390.073,A -85,B 0,C 180,E1 -24596.456,E2 -24596.456} C_VEL
LIN {X 0,Y 147.262,Z 385.725,A -85,B 0,C 180,E1 -24601.67,E2 -24601.67} C_VEL
LIN {X 0,Y 153.763,Z 379.855,A -85,B 0,C 180,E1 -24606.459,E2 -24606.459} C_VEL
LIN {X 0,Y 160.321,Z 373.289,A -85,B 0,C 180,E1 -24610.29,E2 -24610.29} C_VEL
LIN {X 0,Y 167.68,Z 365.176,A -85,B 0,C 180,E1 -24613.759,E2 -24613.759} C_VEL
LIN {X 0,Y 174.936,Z 355.884,A -85,B 0,C 180,E1 -24616.773,E2 -24616.773} C_VEL
LIN {X 0,Y 181.436,Z 346.575,A -85,B 0,C 180,E1 -24619.059,E2 -24619.059} C_VEL
LIN {X 0,Y 188.331,Z 335.231,A -85,B 0,C 180,E1 -24621.173,E2 -24621.173} C_VEL
LIN {X 0,Y 194.088,Z 324.004,A -85,B 0,C 180,E1 -24622.814,E2 -24622.814} C_VEL
LIN {X 0,Y 199.46,Z 311.732,A -85,B 0,C 180,E1 -24624.14,E2 -24624.14} C_VEL
LIN {X 0,Y 204.25,Z 298.094,A -85,B 0,C 180,E1 -24625.241,E2 -24625.241} C_VEL
LIN {X 0,Y 207.942,Z 284.18,A -85,B 0,C 180,E1 -24626.061,E2 -24626.061} C_VEL
LIN {X 0,Y 210.537,Z 269.889,A -85,B 0,C 180,E1 -24626.652,E2 -24626.652} C_VEL
LIN {X 0,Y 213.833,Z 236.332,A -85,B 0,C 180,E1 -24627.554,E2 -24627.554} C_VEL
LIN {X 0,Y 210.721,Z 228.183,A -85,B 0,C 180,E1 -24630.091,E2 -24630.091} C_VEL
LIN {X 0,Y 207.643,Z 220.904,A -85,B 0,C 180,E1 -24632.925,E2 -24632.925} C_VEL
LIN {X 0,Y 204.853,Z 214.628,A -85,B 0,C 180,E1 -24635.932,E2 -24635.932} C_VEL
LIN {X 0,Y 202.015,Z 209.088,A -85,B 0,C 180,E1 -24639.635,E2 -24639.635} C_VEL
LIN {X 0,Y 199.947,Z 205.292,A -85,B 0,C 180,E1 -24643.392,E2 -24643.392} C_VEL
LIN {X 0,Y 198.017,Z 201.018,A -85,B 0,C 180,E1 -24651.567,E2 -24651.567} C_VEL
LIN {X 0,Y 198.084,Z 201.153,A -85,B 0,C 180,E1 -24653.883,E2 -24653.883} C_VEL
LIN {X 0,Y 198.615,Z 202.803,A -85,B 0,C 180,E1 -24657.267,E2 -24657.267} C_VEL
LIN {X 0,Y 200.522,Z 205.856,A -85,B 0,C 180,E1 -24662.118,E2 -24662.118} C_VEL
LIN {X 0,Y 202.818,Z 209.933,A -85,B 0,C 180,E1 -24665.839,E2 -24665.839} C_VEL
LIN {X 0,Y 205.538,Z 214.591,A -85,B 0,C 180,E1 -24669.099,E2 -24669.099} C_VEL
LIN {X 0,Y 208.225,Z 219.372,A -85,B 0,C 180,E1 -24671.777,E2 -24671.777} C_VEL
LIN {X 0,Y 211.883,Z 226.146,A -85,B 0,C 180,E1 -24674.889,E2 -24674.889} C_VEL
LIN {X 0,Y 214.237,Z 231.237,A -85,B 0,C 180,E1 -24676.7,E2 -24676.7} C_VEL
LIN {X 0,Y 210.954,Z 264.89,A -85,B 0,C 180,E1 -24677.628,E2 -24677.628} C_VEL
LIN {X 0,Y 208.35,Z 279.292,A -85,B 0,C 180,E1 -24678.251,E2 -24678.251} C_VEL
LIN {X 0,Y 204.946,Z 292.343,A -85,B 0,C 180,E1 -24679.054,E2 -24679.054} C_VEL
LIN {X 0,Y 200.819,Z 304.796,A -85,B 0,C 180,E1 -24680.135,E2 -24680.135} C_VEL
LIN {X 0,Y 195.582,Z 317.493,A -85,B 0,C 180,E1 -24681.592,E2 -24681.592} C_VEL
LIN {X 0,Y 189.5,Z 329.548,A -85,B 0,C 180,E1 -24683.373,E2 -24683.373} C_VEL
LIN {X 0,Y 182.968,Z 340.504,A -85,B 0,C 180,E1 -24685.484,E2 -24685.484} C_VEL
LIN {X 0,Y 176.698,Z 349.597,A -85,B 0,C 180,E1 -24687.746,E2 -24687.746} C_VEL
LIN {X 0,Y 169.569,Z 358.696,A -85,B 0,C 180,E1 -24690.676,E2 -24690.676} C_VEL
LIN {X 0,Y 162.214,Z 366.977,A -85,B 0,C 180,E1 -24694.268,E2 -24694.268} C_VEL
LIN {X 0,Y 155.902,Z 373.233,A -85,B 0,C 180,E1 -24697.912,E2 -24697.912} C_VEL
LIN {X 0,Y 150.545,Z 378.015,A -85,B 0,C 180,E1 -24701.669,E2 -24701.669} C_VEL
LIN {X 0,Y 144.717,Z 382.638,A -85,B 0,C 180,E1 -24706.742,E2 -24706.742} C_VEL
LIN {X 0,Y 141.836,Z 384.628,A -85,B 0,C 180,E1 -24709.893,E2 -24709.893} C_VEL
LIN {X 0,Y 137.717,Z 387.028,A -85,B 0,C 180,E1 -24715.846,E2 -24715.846} C_VEL
LIN {X 0,Y 134.835,Z 387.969,A -85,B 0,C 180,E1 -24722.361,E2 -24722.361} C_VEL
LIN {X 0,Y 133.433,Z 387.446,A -85,B 0,C 180,E1 -24728.36,E2 -24728.36} C_VEL
LIN {X 0,Y 133.107,Z 386.573,A -85,B 0,C 180,E1 -24731.839,E2 -24731.839} C_VEL
LIN {X 0,Y 133.098,Z 384.021,A -85,B 0,C 180,E1 -24737.802,E2 -24737.802} C_VEL
LIN {X 0,Y 133.755,Z 381.04,A -85,B 0,C 180,E1 -24742.448,E2 -24742.448} C_VEL
LIN {X 0,Y 134.839,Z 377.227,A -85,B 0,C 180,E1 -24747.008,E2 -24747.008} C_VEL
LIN {X 0,Y 136.373,Z 372.515,A -85,B 0,C 180,E1 -24751.472,E2 -24751.472} C_VEL
LIN {X 0,Y 139.014,Z 365.65,A -85,B 0,C 180,E1 -24756.527,E2 -24756.527} C_VEL
LIN {X 0,Y 142.559,Z 357.119,A -85,B 0,C 180,E1 -24761.369,E2 -24761.369} C_VEL
LIN {X 0,Y 146.37,Z 347.867,A -85,B 0,C 180,E1 -24765.464,E2 -24765.464} C_VEL
LIN {X 0,Y 150.185,Z 337.509,A -85,B 0,C 180,E1 -24769.117,E2 -24769.117} C_VEL
LIN {X 0,Y 154.346,Z 326.562,A -85,B 0,C 180,E1 -24772.061,E2 -24772.061} C_VEL
LIN {X 0,Y 158.171,Z 314.637,A -85,B 0,C 180,E1 -24774.613,E2 -24774.613} C_VEL
LIN {X 0,Y 161.818,Z 301.441,A -85,B 0,C 180,E1 -24776.778,E2 -24776.778} C_VEL
LIN {X 0,Y 164.865,Z 287.479,A -85,B 0,C 180,E1 -24778.48,E2 -24778.48} C_VEL
LIN {X 0,Y 167.111,Z 273.598,A -85,B 0,C 180,E1 -24779.697,E2 -24779.697} C_VEL
LIN {X 0,Y 168.662,Z 260.114,A -85,B 0,C 180,E1 -24780.459,E2 -24780.459} C_VEL
LIN {X 0,Y 172.996,Z 198.393,A -85,B 0,C 180,E1 -24782.677,E2 -24782.677} C_VEL
LIN {X 0,Y 168.055,Z 187.755,A -85,B 0,C 180,E1 -24784.847,E2 -24784.847} C_VEL
LIN {X 0,Y 163.03,Z 178.229,A -85,B 0,C 180,E1 -24787.2,E2 -24787.2} C_VEL
LIN {X 0,Y 157.62,Z 169.135,A -85,B 0,C 180,E1 -24789.952,E2 -24789.952} C_VEL
LIN {X 0,Y 152.745,Z 161.695,A -85,B 0,C 180,E1 -24792.692,E2 -24792.692} C_VEL
LIN {X 0,Y 150.08,Z 157.979,A -85,B 0,C 180,E1 -24794.303,E2 -24794.303} C_VEL
LIN {X 0,Y 147.288,Z 154.084,A -85,B 0,C 180,E1 -24796.117,E2 -24796.117} C_VEL
LIN {X 0,Y 144.804,Z 150.738,A -85,B 0,C 180,E1 -24797.853,E2 -24797.853} C_VEL
LIN {X 0,Y 143.978,Z 149.729,A -85,B 0,C 180,E1 -24798.453,E2 -24798.453} C_VEL
LIN {X 0,Y 141.47,Z 146.93,A -85,B 0,C 180,E1 -24800.357,E2 -24800.357} C_VEL
LIN {X 0,Y 140.397,Z 144.783,A -85,B 0,C 180,E1 -24801.323,E2 -24801.323} C_VEL
LIN {X 0,Y 137.745,Z 142.925,A -85,B 0,C 180,E1 -24803.521,E2 -24803.521} C_VEL
LIN {X 0,Y 136.299,Z 140.341,A -85,B 0,C 180,E1 -24805.009,E2 -24805.009} C_VEL
LIN {X 0,Y 136.06,Z 139.151,A -85,B 0,C 180,E1 -24805.389,E2 -24805.389} C_VEL
LIN {X 0,Y 136.127,Z 139.105,A -85,B 0,C 180,E1 -24812.324,E2 -24812.324} C_VEL
LIN {X 0,Y 136.26,Z 139.127,A -85,B 0,C 180,E1 -24818.847,E2 -24818.847} C_VEL
LIN {X 0,Y 136.279,Z 139.121,A -85,B 0,C 180,E1 -24825.068,E2 -24825.068} C_VEL
LIN {X 0,Y 136.488,Z 139.107,A -85,B 0,C 180,E1 -24828.124,E2 -24828.124} C_VEL
LIN {X 0,Y 136.593,Z 139.06,A -85,B 0,C 180,E1 -24831.131,E2 -24831.131} C_VEL
LIN {X 0,Y 137.125,Z 139.026,A -85,B 0,C 180,E1 -24840.01,E2 -24840.01} C_VEL
LIN {X 0,Y 136.586,Z 139.091,A -85,B 0,C 180,E1 -24848.889,E2 -24848.889} C_VEL
LIN {X 0,Y 136.486,Z 139.099,A -85,B 0,C 180,E1 -24851.964,E2 -24851.964} C_VEL
LIN {X 0,Y 136.229,Z 139.184,A -85,B 0,C 180,E1 -24858.43,E2 -24858.43} C_VEL
LIN {X 0,Y 136.94,Z 141.459,A -85,B 0,C 180,E1 -24859.302,E2 -24859.302} C_VEL
LIN {X 0,Y 138.958,Z 143.872,A -85,B 0,C 180,E1 -24861.166,E2 -24861.166} C_VEL
LIN {X 0,Y 140.517,Z 145.041,A -85,B 0,C 180,E1 -24862.428,E2 -24862.428} C_VEL
LIN {X 0,Y 142.308,Z 148.106,A -85,B 0,C 180,E1 -24863.956,E2 -24863.956} C_VEL
LIN {X 0,Y 144.642,Z 150.456,A -85,B 0,C 180,E1 -24865.651,E2 -24865.651} C_VEL
LIN {X 0,Y 147.105,Z 153.969,A -85,B 0,C 180,E1 -24867.395,E2 -24867.395} C_VEL
LIN {X 0,Y 148.436,Z 155.62,A -85,B 0,C 180,E1 -24868.269,E2 -24868.269} C_VEL
LIN {X 0,Y 151.985,Z 160.67,A -85,B 0,C 180,E1 -24870.499,E2 -24870.499} C_VEL
LIN {X 0,Y 156.561,Z 167.462,A -85,B 0,C 180,E1 -24873.102,E2 -24873.102} C_VEL
LIN {X 0,Y 161.203,Z 175.205,A -85,B 0,C 180,E1 -24875.53,E2 -24875.53} C_VEL
LIN {X 0,Y 167.027,Z 188.634,A -85,B 0,C 180,E1 -24878.481,E2 -24878.481} C_VEL
LIN {X 0,Y 171.379,Z 200.792,A -85,B 0,C 180,E1 -24880.59,E2 -24880.59} C_VEL
LIN {X 0,Y 172.712,Z 204.919,A -85,B 0,C 180,E1 -24881.226,E2 -24881.226} C_VEL
LIN {X 0,Y 168.256,Z 270.265,A -85,B 0,C 180,E1 -24883.657,E2 -24883.657} C_VEL
LIN {X 0,Y 166.269,Z 285.162,A -85,B 0,C 180,E1 -24884.61,E2 -24884.61} C_VEL
LIN {X 0,Y 163.823,Z 297.986,A -85,B 0,C 180,E1 -24885.809,E2 -24885.809} C_VEL
LIN {X 0,Y 160.822,Z 310.353,A -85,B 0,C 180,E1 -24887.368,E2 -24887.368} C_VEL
LIN {X 0,Y 157.733,Z 320.938,A -85,B 0,C 180,E1 -24889.067,E2 -24889.067} C_VEL
LIN {X 0,Y 153.978,Z 332.762,A -85,B 0,C 180,E1 -24891.551,E2 -24891.551} C_VEL
LIN {X 0,Y 151.343,Z 339.684,A -85,B 0,C 180,E1 -24893.287,E2 -24893.287} C_VEL
LIN {X 0,Y 147.876,Z 348.802,A -85,B 0,C 180,E1 -24896.057,E2 -24896.057} C_VEL
LIN {X 0,Y 143.731,Z 358.924,A -85,B 0,C 180,E1 -24899.926,E2 -24899.926} C_VEL
LIN {X 0,Y 140.304,Z 367.445,A -85,B 0,C 180,E1 -24904.091,E2 -24904.091} C_VEL
LIN {X 0,Y 137.282,Z 375.319,A -85,B 0,C 180,E1 -24909.005,E2 -24909.005} C_VEL
LIN {X 0,Y 135.56,Z 380.342,A -85,B 0,C 180,E1 -24912.938,E2 -24912.938} C_VEL
LIN {X 0,Y 134.144,Z 382.819,A -85,B 0,C 180,E1 -24915.142,E2 -24915.142} C_VEL
LIN {X 0,Y 130.43,Z 386.249,A -85,B 0,C 180,E1 -24918.835,E2 -24918.835} C_VEL
LIN {X 0,Y 127.611,Z 388.571,A -85,B 0,C 180,E1 -24921.993,E2 -24921.993} C_VEL
LIN {X 0,Y 126.423,Z 390.13,A -85,B 0,C 180,E1 -24924.531,E2 -24924.531} C_VEL
LIN {X 0,Y 126.317,Z 390.591,A -85,B 0,C 180,E1 -24925.403,E2 -24925.403} C_VEL
LIN {X 0,Y 126.464,Z 392.746,A -85,B 0,C 180,E1 -24930.005,E2 -24930.005} C_VEL
LIN {X 0,Y 126.388,Z 393.763,A -85,B 0,C 180,E1 -24933.192,E2 -24933.192} C_VEL
LIN {X 0,Y 126.732,Z 394.788,A -85,B 0,C 180,E1 -24939.581,E2 -24939.581} C_VEL
LIN {X 0,Y 128.253,Z 394.517,A -85,B 0,C 180,E1 -24945.906,E2 -24945.906} C_VEL
LIN {X 0,Y 131.272,Z 392.962,A -85,B 0,C 180,E1 -24952.014,E2 -24952.014} C_VEL
LIN {X 0,Y 135.628,Z 390.091,A -85,B 0,C 180,E1 -24957.803,E2 -24957.803} C_VEL
LIN {X 0,Y 141.248,Z 385.826,A -85,B 0,C 180,E1 -24963.188,E2 -24963.188} C_VEL
LIN {X 0,Y 148.103,Z 380.044,A -85,B 0,C 180,E1 -24968.094,E2 -24968.094} C_VEL
LIN {X 0,Y 154.982,Z 373.573,A -85,B 0,C 180,E1 -24971.985,E2 -24971.985} C_VEL
LIN {X 0,Y 162.641,Z 365.577,A -85,B 0,C 180,E1 -24975.484,E2 -24975.484} C_VEL
LIN {X 0,Y 169.954,Z 356.732,A -85,B 0,C 180,E1 -24978.424,E2 -24978.424} C_VEL
LIN {X 0,Y 176.887,Z 347.269,A -85,B 0,C 180,E1 -24980.788,E2 -24980.788} C_VEL
LIN {X 0,Y 183.992,Z 336.147,A -85,B 0,C 180,E1 -24982.884,E2 -24982.884} C_VEL
LIN {X 0,Y 189.922,Z 325.151,A -85,B 0,C 180,E1 -24984.503,E2 -24984.503} C_VEL
LIN {X 0,Y 195.434,Z 313.199,A -85,B 0,C 180,E1 -24985.807,E2 -24985.807} C_VEL
LIN {X 0,Y 200.324,Z 300.046,A -85,B 0,C 180,E1 -24986.893,E2 -24986.893} C_VEL
LIN {X 0,Y 204.334,Z 285.974,A -85,B 0,C 180,E1 -24987.736,E2 -24987.736} C_VEL
LIN {X 0,Y 207.033,Z 272.419,A -85,B 0,C 180,E1 -24988.325,E2 -24988.325} C_VEL
LIN {X 0,Y 209.324,Z 252.534,A -85,B 0,C 180,E1 -24988.875,E2 -24988.875} C_VEL
LIN {X 0,Y 210.538,Z 239.507,A -85,B 0,C 180,E1 -24989.228,E2 -24989.228} C_VEL
LIN {X 0,Y 207.178,Z 230.519,A -85,B 0,C 180,E1 -24992.312,E2 -24992.312} C_VEL
LIN {X 0,Y 204.111,Z 223.152,A -85,B 0,C 180,E1 -24995.589,E2 -24995.589} C_VEL
LIN {X 0,Y 202.514,Z 219.737,A -85,B 0,C 180,E1 -24997.552,E2 -24997.552} C_VEL
LIN {X 0,Y 200.623,Z 215.609,A -85,B 0,C 180,E1 -25000.338,E2 -25000.338} C_VEL
LIN {X 0,Y 198.847,Z 212.18,A -85,B 0,C 180,E1 -25003.808,E2 -25003.808} C_VEL
LIN {X 0,Y 197.125,Z 208.038,A -85,B 0,C 180,E1 -25011.795,E2 -25011.795} C_VEL
LIN {X 0,Y 197.258,Z 208.534,A -85,B 0,C 180,E1 -25014.622,E2 -25014.622} C_VEL
LIN {X 0,Y 199.354,Z 212.646,A -85,B 0,C 180,E1 -25021.622,E2 -25021.622} C_VEL
LIN {X 0,Y 201.53,Z 216.801,A -85,B 0,C 180,E1 -25025.39,E2 -25025.39} C_VEL
LIN {X 0,Y 203.824,Z 220.893,A -85,B 0,C 180,E1 -25028.298,E2 -25028.298} C_VEL
LIN {X 0,Y 206.844,Z 226.41,A -85,B 0,C 180,E1 -25031.446,E2 -25031.446} C_VEL
LIN {X 0,Y 210.648,Z 234.064,A -85,B 0,C 180,E1 -25034.793,E2 -25034.793} C_VEL
LIN {X 0,Y 210.924,Z 234.692,A -85,B 0,C 180,E1 -25035.02,E2 -25035.02} C_VEL
LIN {X 0,Y 207.815,Z 265.502,A -85,B 0,C 180,E1 -25035.892,E2 -25035.892} C_VEL
LIN {X 0,Y 205.037,Z 280.17,A -85,B 0,C 180,E1 -25036.521,E2 -25036.521} C_VEL
LIN {X 0,Y 201.532,Z 293.091,A -85,B 0,C 180,E1 -25037.314,E2 -25037.314} C_VEL
LIN {X 0,Y 196.909,Z 306.38,A -85,B 0,C 180,E1 -25038.472,E2 -25038.472} C_VEL
LIN {X 0,Y 191.54,Z 318.749,A -85,B 0,C 180,E1 -25039.902,E2 -25039.902} C_VEL
LIN {X 0,Y 185.281,Z 330.614,A -85,B 0,C 180,E1 -25041.663,E2 -25041.663} C_VEL
LIN {X 0,Y 178.352,Z 341.68,A -85,B 0,C 180,E1 -25043.81,E2 -25043.81} C_VEL
LIN {X 0,Y 171.09,Z 351.644,A -85,B 0,C 180,E1 -25046.378,E2 -25046.378} C_VEL
LIN {X 0,Y 163.465,Z 360.689,A -85,B 0,C 180,E1 -25049.462,E2 -25049.462} C_VEL
LIN {X 0,Y 157.229,Z 367.294,A -85,B 0,C 180,E1 -25052.427,E2 -25052.427} C_VEL
LIN {X 0,Y 151.358,Z 372.826,A -85,B 0,C 180,E1 -25055.646,E2 -25055.646} C_VEL
LIN {X 0,Y 145.616,Z 377.731,A -85,B 0,C 180,E1 -25059.44,E2 -25059.44} C_VEL
LIN {X 0,Y 140.496,Z 381.62,A -85,B 0,C 180,E1 -25063.498,E2 -25063.498} C_VEL
LIN {X 0,Y 136.108,Z 384.582,A -85,B 0,C 180,E1 -25067.83,E2 -25067.83} C_VEL
LIN {X 0,Y 131.508,Z 387.098,A -85,B 0,C 180,E1 -25073.99,E2 -25073.99} C_VEL
LIN {X 0,Y 128.315,Z 388.135,A -85,B 0,C 180,E1 -25080.461,E2 -25080.461} C_VEL
LIN {X 0,Y 126.516,Z 387.732,A -85,B 0,C 180,E1 -25087.112,E2 -25087.112} C_VEL
LIN {X 0,Y 126.047,Z 386.758,A -85,B 0,C 180,E1 -25091.379,E2 -25091.379} C_VEL
LIN {X 0,Y 125.94,Z 384.471,A -85,B 0,C 180,E1 -25097.097,E2 -25097.097} C_VEL
LIN {X 0,Y 126.575,Z 381.589,A -85,B 0,C 180,E1 -25102.016,E2 -25102.016} C_VEL
LIN {X 0,Y 127.668,Z 377.888,A -85,B 0,C 180,E1 -25106.84,E2 -25106.84} C_VEL
LIN {X 0,Y 129.218,Z 373.255,A -85,B 0,C 180,E1 -25111.554,E2 -25111.554} C_VEL
LIN {X 0,Y 131.925,Z 366.549,A -85,B 0,C 180,E1 -25116.88,E2 -25116.88} C_VEL
LIN {X 0,Y 135.561,Z 358.193,A -85,B 0,C 180,E1 -25121.964,E2 -25121.964} C_VEL
LIN {X 0,Y 139.63,Z 348.766,A -85,B 0,C 180,E1 -25126.393,E2 -25126.393} C_VEL
LIN {X 0,Y 143.491,Z 338.962,A -85,B 0,C 180,E1 -25130.046,E2 -25130.046} C_VEL
LIN {X 0,Y 147.709,Z 328.29,A -85,B 0,C 180,E1 -25133.108,E2 -25133.108} C_VEL
LIN {X 0,Y 151.741,Z 316.669,A -85,B 0,C 180,E1 -25135.731,E2 -25135.731} C_VEL
LIN {X 0,Y 155.524,Z 303.917,A -85,B 0,C 180,E1 -25137.955,E2 -25137.955} C_VEL
LIN {X 0,Y 158.695,Z 290.742,A -85,B 0,C 180,E1 -25139.695,E2 -25139.695} C_VEL
LIN {X 0,Y 161.3,Z 276.525,A -85,B 0,C 180,E1 -25141.063,E2 -25141.063} C_VEL
LIN {X 0,Y 163.004,Z 263.142,A -85,B 0,C 180,E1 -25141.923,E2 -25141.923} C_VEL
LIN {X 0,Y 167.616,Z 200.58,A -85,B 0,C 180,E1 -25144.229,E2 -25144.229} C_VEL
LIN {X 0,Y 162.197,Z 188.935,A -85,B 0,C 180,E1 -25146.822,E2 -25146.822} C_VEL
LIN {X 0,Y 155.907,Z 177.38,A -85,B 0,C 180,E1 -25150.102,E2 -25150.102} C_VEL
LIN {X 0,Y 149.998,Z 167.9,A -85,B 0,C 180,E1 -25153.554,E2 -25153.554} C_VEL
LIN {X 0,Y 146.943,Z 163.574,A -85,B 0,C 180,E1 -25155.503,E2 -25155.503} C_VEL
LIN {X 0,Y 144.387,Z 159.941,A -85,B 0,C 180,E1 -25157.274,E2 -25157.274} C_VEL
LIN {X 0,Y 141.338,Z 155.81,A -85,B 0,C 180,E1 -25159.572,E2 -25159.572} C_VEL
LIN {X 0,Y 138.704,Z 152.529,A -85,B 0,C 180,E1 -25161.738,E2 -25161.738} C_VEL
LIN {X 0,Y 137.851,Z 151.151,A -85,B 0,C 180,E1 -25162.525,E2 -25162.525} C_VEL
LIN {X 0,Y 135.316,Z 148.867,A -85,B 0,C 180,E1 -25164.831,E2 -25164.831} C_VEL
LIN {X 0,Y 133.57,Z 145.812,A -85,B 0,C 180,E1 -25166.775,E2 -25166.775} C_VEL
LIN {X 0,Y 130.803,Z 143.92,A -85,B 0,C 180,E1 -25169.878,E2 -25169.878} C_VEL
LIN {X 0,Y 129.494,Z 141.665,A -85,B 0,C 180,E1 -25171.771,E2 -25171.771} C_VEL
LIN {X 0,Y 129.062,Z 139.985,A -85,B 0,C 180,E1 -25172.66,E2 -25172.66} C_VEL
LIN {X 0,Y 129.113,Z 140.024,A -85,B 0,C 180,E1 -25177.71,E2 -25177.71} C_VEL
LIN {X 0,Y 129.169,Z 140.011,A -85,B 0,C 180,E1 -25180.958,E2 -25180.958} C_VEL
LIN {X 0,Y 129.404,Z 139.989,A -85,B 0,C 180,E1 -25187.824,E2 -25187.824} C_VEL
LIN {X 0,Y 129.516,Z 139.946,A -85,B 0,C 180,E1 -25190.642,E2 -25190.642} C_VEL
LIN {X 0,Y 130.08,Z 139.902,A -85,B 0,C 180,E1 -25200.01,E2 -25200.01} C_VEL
LIN {X 0,Y 129.511,Z 139.976,A -85,B 0,C 180,E1 -25209.379,E2 -25209.379} C_VEL
LIN {X 0,Y 129.476,Z 140.094,A -85,B 0,C 180,E1 -25211.565,E2 -25211.565} C_VEL
LIN {X 0,Y 130.215,Z 142.615,A -85,B 0,C 180,E1 -25212.874,E2 -25212.874} C_VEL
LIN {X 0,Y 132.071,Z 144.867,A -85,B 0,C 180,E1 -25215.243,E2 -25215.243} C_VEL
LIN {X 0,Y 133.989,Z 145.971,A -85,B 0,C 180,E1 -25217.268,E2 -25217.268} C_VEL
LIN {X 0,Y 135.552,Z 148.916,A -85,B 0,C 180,E1 -25219.016,E2 -25219.016} C_VEL
LIN {X 0,Y 138.165,Z 151.529,A -85,B 0,C 180,E1 -25221.394,E2 -25221.394} C_VEL
LIN {X 0,Y 140.588,Z 155.097,A -85,B 0,C 180,E1 -25223.493,E2 -25223.493} C_VEL
LIN {X 0,Y 142.071,Z 156.731,A -85,B 0,C 180,E1 -25224.63,E2 -25224.63} C_VEL
LIN {X 0,Y 144.93,Z 160.536,A -85,B 0,C 180,E1 -25226.725,E2 -25226.725} C_VEL
LIN {X 0,Y 150.719,Z 169.045,A -85,B 0,C 180,E1 -25230.528,E2 -25230.528} C_VEL
LIN {X 0,Y 156.988,Z 179.357,A -85,B 0,C 180,E1 -25234.117,E2 -25234.117} C_VEL
LIN {X 0,Y 162.577,Z 192.693,A -85,B 0,C 180,E1 -25237.177,E2 -25237.177} C_VEL
LIN {X 0,Y 166.482,Z 203.972,A -85,B 0,C 180,E1 -25239.222,E2 -25239.222} C_VEL
LIN {X 0,Y 167.417,Z 207.192,A -85,B 0,C 180,E1 -25239.719,E2 -25239.719} C_VEL
LIN {X 0,Y 162.836,Z 270.24,A -85,B 0,C 180,E1 -25242.08,E2 -25242.08} C_VEL
LIN {X 0,Y 160.905,Z 284.335,A -85,B 0,C 180,E1 -25242.984,E2 -25242.984} C_VEL
LIN {X 0,Y 158.229,Z 297.892,A -85,B 0,C 180,E1 -25244.263,E2 -25244.263} C_VEL
LIN {X 0,Y 154.549,Z 312.006,A -85,B 0,C 180,E1 -25246.099,E2 -25246.099} C_VEL
LIN {X 0,Y 150.463,Z 325.02,A -85,B 0,C 180,E1 -25248.397,E2 -25248.397} C_VEL
LIN {X 0,Y 147.469,Z 333.801,A -85,B 0,C 180,E1 -25250.406,E2 -25250.406} C_VEL
LIN {X 0,Y 144.413,Z 341.72,A -85,B 0,C 180,E1 -25252.537,E2 -25252.537} C_VEL
LIN {X 0,Y 140.383,Z 351.357,A -85,B 0,C 180,E1 -25255.727,E2 -25255.727} C_VEL
LIN {X 0,Y 136.288,Z 361.037,A -85,B 0,C 180,E1 -25259.821,E2 -25259.821} C_VEL
LIN {X 0,Y 132.982,Z 368.757,A -85,B 0,C 180,E1 -25263.972,E2 -25263.972} C_VEL
LIN {X 0,Y 129.859,Z 376.681,A -85,B 0,C 180,E1 -25269.409,E2 -25269.409} C_VEL
LIN {X 0,Y 127.963,Z 381.949,A -85,B 0,C 180,E1 -25274.066,E2 -25274.066} C_VEL
LIN {X 0,Y 126.913,Z 386.231,A -85,B 0,C 180,E1 -25278.829,E2 -25278.829} C_VEL
LIN {X 0,Y 126.416,Z 389.617,A -85,B 0,C 180,E1 -25283.621,E2 -25283.621} C_VEL
LIN {X 0,Y 126.317,Z 390.591,A -85,B 0,C 180,E1 -25285.403,E2 -25285.403} C_VEL
LIN {X 0,Y 125.582,Z 391.878,A -85,B 0,C 180,E1 -25288,E2 -25288} C_VEL
LIN {X 0,Y 123.946,Z 392.848,A -85,B 0,C 180,E1 -25290.589,E2 -25290.589} C_VEL
LIN {X 0,Y 120.348,Z 394.1,A -85,B 0,C 180,E1 -25295.959,E2 -25295.959} C_VEL
LIN {X 0,Y 119.587,Z 394.449,A -85,B 0,C 180,E1 -25298.803,E2 -25298.803} C_VEL
LIN {X 0,Y 119.643,Z 394.527,A -85,B 0,C 180,E1 -25299.761,E2 -25299.761} C_VEL
LIN {X 0,Y 120.417,Z 394.636,A -85,B 0,C 180,E1 -25303.505,E2 -25303.505} C_VEL
LIN {X 0,Y 122.826,Z 393.799,A -85,B 0,C 180,E1 -25310.084,E2 -25310.084} C_VEL
LIN {X 0,Y 126.842,Z 391.671,A -85,B 0,C 180,E1 -25316.317,E2 -25316.317} C_VEL
LIN {X 0,Y 132.168,Z 388.198,A -85,B 0,C 180,E1 -25322.128,E2 -25322.128} C_VEL
LIN {X 0,Y 138.807,Z 383.278,A -85,B 0,C 180,E1 -25327.419,E2 -25327.419} C_VEL
LIN {X 0,Y 146.58,Z 376.769,A -85,B 0,C 180,E1 -25332.168,E2 -25332.168} C_VEL
LIN {X 0,Y 154.264,Z 369.562,A -85,B 0,C 180,E1 -25335.857,E2 -25335.857} C_VEL
LIN {X 0,Y 162.551,Z 360.693,A -85,B 0,C 180,E1 -25339.173,E2 -25339.173} C_VEL
LIN {X 0,Y 169.915,Z 351.456,A -85,B 0,C 180,E1 -25341.807,E2 -25341.807} C_VEL
LIN {X 0,Y 177.825,Z 340.203,A -85,B 0,C 180,E1 -25344.12,E2 -25344.12} C_VEL
LIN {X 0,Y 184.546,Z 328.818,A -85,B 0,C 180,E1 -25345.929,E2 -25345.929} C_VEL
LIN {X 0,Y 190.865,Z 316.202,A -85,B 0,C 180,E1 -25347.389,E2 -25347.389} C_VEL
LIN {X 0,Y 195.845,Z 303.967,A -85,B 0,C 180,E1 -25348.466,E2 -25348.466} C_VEL
LIN {X 0,Y 200.258,Z 290.242,A -85,B 0,C 180,E1 -25349.344,E2 -25349.344} C_VEL
LIN {X 0,Y 203.641,Z 275.714,A -85,B 0,C 180,E1 -25349.999,E2 -25349.999} C_VEL
LIN {X 0,Y 205.663,Z 261.446,A -85,B 0,C 180,E1 -25350.445,E2 -25350.445} C_VEL
LIN {X 0,Y 207.438,Z 242.871,A -85,B 0,C 180,E1 -25350.949,E2 -25350.949} C_VEL
LIN {X 0,Y 204.625,Z 235.06,A -85,B 0,C 180,E1 -25353.812,E2 -25353.812} C_VEL
LIN {X 0,Y 202.059,Z 228.535,A -85,B 0,C 180,E1 -25356.855,E2 -25356.855} C_VEL
LIN {X 0,Y 199.519,Z 222.676,A -85,B 0,C 180,E1 -25360.605,E2 -25360.605} C_VEL
LIN {X 0,Y 197.874,Z 219.196,A -85,B 0,C 180,E1 -25363.966,E2 -25363.966} C_VEL
LIN {X 0,Y 196.226,Z 215.218,A -85,B 0,C 180,E1 -25371.757,E2 -25371.757} C_VEL
LIN {X 0,Y 196.375,Z 215.641,A -85,B 0,C 180,E1 -25374.682,E2 -25374.682} C_VEL
LIN {X 0,Y 198.248,Z 219.591,A -85,B 0,C 180,E1 -25381.237,E2 -25381.237} C_VEL
LIN {X 0,Y 200.253,Z 223.628,A -85,B 0,C 180,E1 -25384.927,E2 -25384.927} C_VEL
LIN {X 0,Y 202.363,Z 227.573,A -85,B 0,C 180,E1 -25387.741,E2 -25387.741} C_VEL
LIN {X 0,Y 205.164,Z 233.007,A -85,B 0,C 180,E1 -25390.822,E2 -25390.822} C_VEL
LIN {X 0,Y 207.85,Z 238.774,A -85,B 0,C 180,E1 -25393.373,E2 -25393.373} C_VEL
LIN {X 0,Y 204.967,Z 265.718,A -85,B 0,C 180,E1 -25394.094,E2 -25394.094} C_VEL
LIN {X 0,Y 202.092,Z 280.448,A -85,B 0,C 180,E1 -25394.702,E2 -25394.702} C_VEL
LIN {X 0,Y 198.312,Z 293.942,A -85,B 0,C 180,E1 -25395.518,E2 -25395.518} C_VEL
LIN {X 0,Y 193.707,Z 306.716,A -85,B 0,C 180,E1 -25396.612,E2 -25396.612} C_VEL
LIN {X 0,Y 188.388,Z 318.593,A -85,B 0,C 180,E1 -25397.946,E2 -25397.946} C_VEL
LIN {X 0,Y 181.945,Z 330.507,A -85,B 0,C 180,E1 -25399.681,E2 -25399.681} C_VEL
LIN {X 0,Y 175.221,Z 340.932,A -85,B 0,C 180,E1 -25401.631,E2 -25401.631} C_VEL
LIN {X 0,Y 167.627,Z 351.099,A -85,B 0,C 180,E1 -25404.146,E2 -25404.146} C_VEL
LIN {X 0,Y 159.875,Z 360.047,A -85,B 0,C 180,E1 -25407.098,E2 -25407.098} C_VEL
LIN {X 0,Y 152.377,Z 367.639,A -85,B 0,C 180,E1 -25410.476,E2 -25410.476} C_VEL
LIN {X 0,Y 144.944,Z 374.222,A -85,B 0,C 180,E1 -25414.477,E2 -25414.477} C_VEL
LIN {X 0,Y 138.988,Z 378.922,A -85,B 0,C 180,E1 -25418.387,E2 -25418.387} C_VEL
LIN {X 0,Y 132.682,Z 383.218,A -85,B 0,C 180,E1 -25423.503,E2 -25423.503} C_VEL
LIN {X 0,Y 127.833,Z 386.029,A -85,B 0,C 180,E1 -25428.715,E2 -25428.715} C_VEL
LIN {X 0,Y 123.416,Z 387.923,A -85,B 0,C 180,E1 -25435.282,E2 -25435.282} C_VEL
LIN {X 0,Y 120.546,Z 388.346,A -85,B 0,C 180,E1 -25442.193,E2 -25442.193} C_VEL
LIN {X 0,Y 119.101,Z 387.337,A -85,B 0,C 180,E1 -25449.26,E2 -25449.26} C_VEL
LIN {X 0,Y 118.848,Z 386.301,A -85,B 0,C 180,E1 -25452.797,E2 -25452.797} C_VEL
LIN {X 0,Y 119.084,Z 383.165,A -85,B 0,C 180,E1 -25459.797,E2 -25459.797} C_VEL
LIN {X 0,Y 119.974,Z 380.054,A -85,B 0,C 180,E1 -25464.637,E2 -25464.637} C_VEL
LIN {X 0,Y 121.449,Z 375.616,A -85,B 0,C 180,E1 -25469.995,E2 -25469.995} C_VEL
LIN {X 0,Y 123.48,Z 370.417,A -85,B 0,C 180,E1 -25474.893,E2 -25474.893} C_VEL
LIN {X 0,Y 126.86,Z 362.967,A -85,B 0,C 180,E1 -25480.368,E2 -25480.368} C_VEL
LIN {X 0,Y 130.487,Z 355.164,A -85,B 0,C 180,E1 -25484.818,E2 -25484.818} C_VEL
LIN {X 0,Y 134.694,Z 345.798,A -85,B 0,C 180,E1 -25489.028,E2 -25489.028} C_VEL
LIN {X 0,Y 138.869,Z 335.476,A -85,B 0,C 180,E1 -25492.695,E2 -25492.695} C_VEL
LIN {X 0,Y 143.448,Z 323.991,A -85,B 0,C 180,E1 -25495.769,E2 -25495.769} C_VEL
LIN {X 0,Y 147.77,Z 311.307,A -85,B 0,C 180,E1 -25498.394,E2 -25498.394} C_VEL
LIN {X 0,Y 151.306,Z 299.005,A -85,B 0,C 180,E1 -25500.335,E2 -25500.335} C_VEL
LIN {X 0,Y 154.351,Z 285.475,A -85,B 0,C 180,E1 -25501.955,E2 -25501.955} C_VEL
LIN {X 0,Y 156.565,Z 272.098,A -85,B 0,C 180,E1 -25503.106,E2 -25503.106} C_VEL
LIN {X 0,Y 158.291,Z 257.326,A -85,B 0,C 180,E1 -25503.877,E2 -25503.877} C_VEL
LIN {X 0,Y 162.382,Z 202.86,A -85,B 0,C 180,E1 -25505.871,E2 -25505.871} C_VEL
LIN {X 0,Y 156.484,Z 190.301,A -85,B 0,C 180,E1 -25508.954,E2 -25508.954} C_VEL
LIN {X 0,Y 150.914,Z 180.144,A -85,B 0,C 180,E1 -25512.159,E2 -25512.159} C_VEL
LIN {X 0,Y 145.003,Z 170.581,A -85,B 0,C 180,E1 -25515.982,E2 -25515.982} C_VEL
LIN {X 0,Y 141.191,Z 165.307,A -85,B 0,C 180,E1 -25518.752,E2 -25518.752} C_VEL
LIN {X 0,Y 138.768,Z 161.886,A -85,B 0,C 180,E1 -25520.717,E2 -25520.717} C_VEL
LIN {X 0,Y 136.057,Z 158.198,A -85,B 0,C 180,E1 -25523.138,E2 -25523.138} C_VEL
LIN {X 0,Y 134.834,Z 156.904,A -85,B 0,C 180,E1 -25524.285,E2 -25524.285} C_VEL
LIN {X 0,Y 132.468,Z 153.987,A -85,B 0,C 180,E1 -25526.753,E2 -25526.753} C_VEL
LIN {X 0,Y 131.655,Z 152.472,A -85,B 0,C 180,E1 -25527.749,E2 -25527.749} C_VEL
LIN {X 0,Y 128.915,Z 150.238,A -85,B 0,C 180,E1 -25531.083,E2 -25531.083} C_VEL
LIN {X 0,Y 127.511,Z 147.541,A -85,B 0,C 180,E1 -25533.342,E2 -25533.342} C_VEL
LIN {X 0,Y 127.272,Z 146.882,A -85,B 0,C 180,E1 -25533.796,E2 -25533.796} C_VEL
LIN {X 0,Y 124.256,Z 145.195,A -85,B 0,C 180,E1 -25539.325,E2 -25539.325} C_VEL
LIN {X 0,Y 122.432,Z 141.949,A -85,B 0,C 180,E1 -25545.891,E2 -25545.891} C_VEL
LIN {X 0,Y 122.351,Z 140.866,A -85,B 0,C 180,E1 -25547.532,E2 -25547.532} C_VEL
LIN {X 0,Y 122.442,Z 140.833,A -85,B 0,C 180,E1 -25550.096,E2 -25550.096} C_VEL
LIN {X 0,Y 122.916,Z 140.904,A -85,B 0,C 180,E1 -25559.192,E2 -25559.192} C_VEL
LIN {X 0,Y 123.129,Z 141.553,A -85,B 0,C 180,E1 -25560.215,E2 -25560.215} C_VEL
LIN {X 0,Y 123.656,Z 143.605,A -85,B 0,C 180,E1 -25562.454,E2 -25562.454} C_VEL
LIN {X 0,Y 125.714,Z 145.981,A -85,B 0,C 180,E1 -25567.236,E2 -25567.236} C_VEL
LIN {X 0,Y 127.693,Z 147.073,A -85,B 0,C 180,E1 -25570.441,E2 -25570.441} C_VEL
LIN {X 0,Y 128.995,Z 149.988,A -85,B 0,C 180,E1 -25572.598,E2 -25572.598} C_VEL
LIN {X 0,Y 131.349,Z 152.191,A -85,B 0,C 180,E1 -25575.527,E2 -25575.527} C_VEL
LIN {X 0,Y 132.135,Z 152.984,A -85,B 0,C 180,E1 -25576.423,E2 -25576.423} C_VEL
LIN {X 0,Y 134.434,Z 156.395,A -85,B 0,C 180,E1 -25578.957,E2 -25578.957} C_VEL
LIN {X 0,Y 135.915,Z 157.969,A -85,B 0,C 180,E1 -25580.364,E2 -25580.364} C_VEL
LIN {X 0,Y 138.558,Z 161.684,A -85,B 0,C 180,E1 -25582.751,E2 -25582.751} C_VEL
LIN {X 0,Y 139.746,Z 163.261,A -85,B 0,C 180,E1 -25583.733,E2 -25583.733} C_VEL
LIN {X 0,Y 143.137,Z 168.053,A -85,B 0,C 180,E1 -25586.341,E2 -25586.341} C_VEL
LIN {X 0,Y 147.258,Z 174.18,A -85,B 0,C 180,E1 -25589.174,E2 -25589.174} C_VEL
LIN {X 0,Y 153.166,Z 184.231,A -85,B 0,C 180,E1 -25592.818,E2 -25592.818} C_VEL
LIN {X 0,Y 158.606,Z 197.796,A -85,B 0,C 180,E1 -25596.021,E2 -25596.021} C_VEL
LIN {X 0,Y 162.205,Z 208.894,A -85,B 0,C 180,E1 -25598.067,E2 -25598.067} C_VEL
LIN {X 0,Y 157.523,Z 270.423,A -85,B 0,C 180,E1 -25600.407,E2 -25600.407} C_VEL
LIN {X 0,Y 155.391,Z 285.04,A -85,B 0,C 180,E1 -25601.372,E2 -25601.372} C_VEL
LIN {X 0,Y 152.757,Z 297.797,A -85,B 0,C 180,E1 -25602.604,E2 -25602.604} C_VEL
LIN {X 0,Y 148.935,Z 311.891,A -85,B 0,C 180,E1 -25604.467,E2 -25604.467} C_VEL
LIN {X 0,Y 144.804,Z 324.514,A -85,B 0,C 180,E1 -25606.732,E2 -25606.732} C_VEL
LIN {X 0,Y 141.544,Z 333.66,A -85,B 0,C 180,E1 -25608.866,E2 -25608.866} C_VEL
LIN {X 0,Y 138.336,Z 341.572,A -85,B 0,C 180,E1 -25611.051,E2 -25611.051} C_VEL
LIN {X 0,Y 133.711,Z 352.104,A -85,B 0,C 180,E1 -25614.684,E2 -25614.684} C_VEL
LIN {X 0,Y 129.467,Z 361.607,A -85,B 0,C 180,E1 -25618.961,E2 -25618.961} C_VEL
LIN {X 0,Y 125.892,Z 369.478,A -85,B 0,C 180,E1 -25623.479,E2 -25623.479} C_VEL
LIN {X 0,Y 123.153,Z 376,A -85,B 0,C 180,E1 -25628.232,E2 -25628.232} C_VEL
LIN {X 0,Y 121.095,Z 381.362,A -85,B 0,C 180,E1 -25633.136,E2 -25633.136} C_VEL
LIN {X 0,Y 119.652,Z 386.992,A -85,B 0,C 180,E1 -25639.856,E2 -25639.856} C_VEL
LIN {X 0,Y 119.225,Z 390.344,A -85,B 0,C 180,E1 -25645.415,E2 -25645.415} C_VEL
LIN {X 0,Y 119.379,Z 392.416,A -85,B 0,C 180,E1 -25650.005,E2 -25650.005} C_VEL
LIN {X 0,Y 119.295,Z 393.471,A -85,B 0,C 180,E1 -25653.382,E2 -25653.382} C_VEL
LIN {X 0,Y 119.643,Z 394.527,A -85,B 0,C 180,E1 -25659.761,E2 -25659.761} C_VEL
LIN {X 0,Y 119.524,Z 394.721,A -85,B 0,C 180,E1 -25662.587,E2 -25662.587} C_VEL
LIN {X 0,Y 118.058,Z 394.492,A -85,B 0,C 180,E1 -25667.317,E2 -25667.317} C_VEL
LIN {X 0,Y 117.289,Z 393.822,A -85,B 0,C 180,E1 -25671.164,E2 -25671.164} C_VEL
LIN {X 0,Y 117.841,Z 393.038,A -85,B 0,C 180,E1 -25674.014,E2 -25674.014} C_VEL
LIN {X 0,Y 118.351,Z 392.723,A -85,B 0,C 180,E1 -25674.927,E2 -25674.927} C_VEL
LIN {X 0,Y 123.171,Z 390.125,A -85,B 0,C 180,E1 -25680.904,E2 -25680.904} C_VEL
LIN {X 0,Y 129.541,Z 386.027,A -85,B 0,C 180,E1 -25686.645,E2 -25686.645} C_VEL
LIN {X 0,Y 137.209,Z 380.421,A -85,B 0,C 180,E1 -25691.755,E2 -25691.755} C_VEL
LIN {X 0,Y 144.724,Z 374.15,A -85,B 0,C 180,E1 -25695.754,E2 -25695.754} C_VEL
LIN {X 0,Y 153.052,Z 366.381,A -85,B 0,C 180,E1 -25699.264,E2 -25699.264} C_VEL
LIN {X 0,Y 160.47,Z 358.322,A -85,B 0,C 180,E1 -25702.035,E2 -25702.035} C_VEL
LIN {X 0,Y 168.335,Z 348.641,A -85,B 0,C 180,E1 -25704.506,E2 -25704.506} C_VEL
LIN {X 0,Y 175.863,Z 337.92,A -85,B 0,C 180,E1 -25706.541,E2 -25706.541} C_VEL
LIN {X 0,Y 182.121,Z 327.378,A -85,B 0,C 180,E1 -25708.105,E2 -25708.105} C_VEL
LIN {X 0,Y 187.909,Z 316.041,A -85,B 0,C 180,E1 -25709.347,E2 -25709.347} C_VEL
LIN {X 0,Y 193.005,Z 303.818,A -85,B 0,C 180,E1 -25710.391,E2 -25710.391} C_VEL
LIN {X 0,Y 197.341,Z 290.724,A -85,B 0,C 180,E1 -25711.204,E2 -25711.204} C_VEL
LIN {X 0,Y 200.778,Z 276.594,A -85,B 0,C 180,E1 -25711.827,E2 -25711.827} C_VEL
LIN {X 0,Y 202.923,Z 262.628,A -85,B 0,C 180,E1 -25712.259,E2 -25712.259} C_VEL
LIN {X 0,Y 204.509,Z 246.411,A -85,B 0,C 180,E1 -25712.717,E2 -25712.717} C_VEL
LIN {X 0,Y 202.177,Z 239.503,A -85,B 0,C 180,E1 -25715.395,E2 -25715.395} C_VEL
LIN {X 0,Y 200.027,Z 233.697,A -85,B 0,C 180,E1 -25718.267,E2 -25718.267} C_VEL
LIN {X 0,Y 198.03,Z 228.917,A -85,B 0,C 180,E1 -25721.597,E2 -25721.597} C_VEL
LIN {X 0,Y 196.692,Z 226.011,A -85,B 0,C 180,E1 -25724.611,E2 -25724.611} C_VEL
LIN {X 0,Y 195.328,Z 222.382,A -85,B 0,C 180,E1 -25731.719,E2 -25731.719} C_VEL
LIN {X 0,Y 195.439,Z 222.555,A -85,B 0,C 180,E1 -25734.229,E2 -25734.229} C_VEL
LIN {X 0,Y 197.11,Z 226.376,A -85,B 0,C 180,E1 -25740.733,E2 -25740.733} C_VEL
LIN {X 0,Y 198.84,Z 230.085,A -85,B 0,C 180,E1 -25744.177,E2 -25744.177} C_VEL
LIN {X 0,Y 201.027,Z 234.497,A -85,B 0,C 180,E1 -25747.315,E2 -25747.315} C_VEL
LIN {X 0,Y 204.077,Z 240.844,A -85,B 0,C 180,E1 -25750.786,E2 -25750.786} C_VEL
LIN {X 0,Y 204.911,Z 242.724,A -85,B 0,C 180,E1 -25751.633,E2 -25751.633} C_VEL
LIN {X 0,Y 202.304,Z 266.027,A -85,B 0,C 180,E1 -25752.246,E2 -25752.246} C_VEL
LIN {X 0,Y 199.417,Z 280.488,A -85,B 0,C 180,E1 -25752.823,E2 -25752.823} C_VEL
LIN {X 0,Y 195.625,Z 293.731,A -85,B 0,C 180,E1 -25753.582,E2 -25753.582} C_VEL
LIN {X 0,Y 190.726,Z 307.021,A -85,B 0,C 180,E1 -25754.688,E2 -25754.688} C_VEL
LIN {X 0,Y 184.706,Z 319.991,A -85,B 0,C 180,E1 -25756.124,E2 -25756.124} C_VEL
LIN {X 0,Y 178.104,Z 331.648,A -85,B 0,C 180,E1 -25757.82,E2 -25757.82} C_VEL
LIN {X 0,Y 171.601,Z 341.302,A -85,B 0,C 180,E1 -25759.605,E2 -25759.605} C_VEL
LIN {X 0,Y 164.632,Z 350.349,A -85,B 0,C 180,E1 -25761.793,E2 -25761.793} C_VEL
LIN {X 0,Y 156.602,Z 359.401,A -85,B 0,C 180,E1 -25764.655,E2 -25764.655} C_VEL
LIN {X 0,Y 148.702,Z 367.125,A -85,B 0,C 180,E1 -25767.953,E2 -25767.953} C_VEL
LIN {X 0,Y 140.783,Z 373.87,A -85,B 0,C 180,E1 -25771.927,E2 -25771.927} C_VEL
LIN {X 0,Y 134.412,Z 378.645,A -85,B 0,C 180,E1 -25775.854,E2 -25775.854} C_VEL
LIN {X 0,Y 128.651,Z 382.401,A -85,B 0,C 180,E1 -25780.105,E2 -25780.105} C_VEL
LIN {X 0,Y 122.211,Z 385.988,A -85,B 0,C 180,E1 -25786.357,E2 -25786.357} C_VEL
LIN {X 0,Y 117.287,Z 388.036,A -85,B 0,C 180,E1 -25793.181,E2 -25793.181} C_VEL
LIN {X 0,Y 113.956,Z 388.579,A -85,B 0,C 180,E1 -25800.431,E2 -25800.431} C_VEL
LIN {X 0,Y 112.163,Z 387.677,A -85,B 0,C 180,E1 -25807.911,E2 -25807.911} C_VEL
LIN {X 0,Y 111.815,Z 386.692,A -85,B 0,C 180,E1 -25811.678,E2 -25811.678} C_VEL
LIN {X 0,Y 111.884,Z 383.663,A -85,B 0,C 180,E1 -25819.133,E2 -25819.133} C_VEL
LIN {X 0,Y 112.886,Z 380.305,A -85,B 0,C 180,E1 -25824.798,E2 -25824.798} C_VEL
LIN {X 0,Y 114.252,Z 376.313,A -85,B 0,C 180,E1 -25829.995,E2 -25829.995} C_VEL
LIN {X 0,Y 116.338,Z 371.203,A -85,B 0,C 180,E1 -25835.194,E2 -25835.194} C_VEL
LIN {X 0,Y 119.839,Z 363.892,A -85,B 0,C 180,E1 -25840.983,E2 -25840.983} C_VEL
LIN {X 0,Y 123.613,Z 356.235,A -85,B 0,C 180,E1 -25845.663,E2 -25845.663} C_VEL
LIN {X 0,Y 128.012,Z 347.051,A -85,B 0,C 180,E1 -25850.063,E2 -25850.063} C_VEL
LIN {X 0,Y 131.886,Z 337.956,A -85,B 0,C 180,E1 -25853.552,E2 -25853.552} C_VEL
LIN {X 0,Y 136.648,Z 326.983,A -85,B 0,C 180,E1 -25856.74,E2 -25856.74} C_VEL
LIN {X 0,Y 141.059,Z 315.017,A -85,B 0,C 180,E1 -25859.467,E2 -25859.467} C_VEL
LIN {X 0,Y 145.204,Z 301.759,A -85,B 0,C 180,E1 -25861.755,E2 -25861.755} C_VEL
LIN {X 0,Y 148.39,Z 289,A -85,B 0,C 180,E1 -25863.402,E2 -25863.402} C_VEL
LIN {X 0,Y 151.112,Z 274.543,A -85,B 0,C 180,E1 -25864.728,E2 -25864.728} C_VEL
LIN {X 0,Y 152.852,Z 261.13,A -85,B 0,C 180,E1 -25865.53,E2 -25865.53} C_VEL
LIN {X 0,Y 157.272,Z 205.275,A -85,B 0,C 180,E1 -25867.62,E2 -25867.62} C_VEL
LIN {X 0,Y 151.905,Z 193.638,A -85,B 0,C 180,E1 -25870.687,E2 -25870.687} C_VEL
LIN {X 0,Y 147.022,Z 184.669,A -85,B 0,C 180,E1 -25873.723,E2 -25873.723} C_VEL
LIN {X 0,Y 141.902,Z 176.097,A -85,B 0,C 180,E1 -25877.303,E2 -25877.303} C_VEL
LIN {X 0,Y 136.51,Z 168.194,A -85,B 0,C 180,E1 -25881.689,E2 -25881.689} C_VEL
LIN {X 0,Y 133.122,Z 163.66,A -85,B 0,C 180,E1 -25884.938,E2 -25884.938} C_VEL
LIN {X 0,Y 130.483,Z 160.366,A -85,B 0,C 180,E1 -25887.843,E2 -25887.843} C_VEL
LIN {X 0,Y 129.676,Z 159.028,A -85,B 0,C 180,E1 -25888.876,E2 -25888.876} C_VEL
LIN {X 0,Y 127.044,Z 156.478,A -85,B 0,C 180,E1 -25892.383,E2 -25892.383} C_VEL
LIN {X 0,Y 125.701,Z 153.746,A -85,B 0,C 180,E1 -25894.779,E2 -25894.779} C_VEL
LIN {X 0,Y 122.704,Z 151.615,A -85,B 0,C 180,E1 -25901.001,E2 -25901.001} C_VEL
LIN {X 0,Y 121.345,Z 148.293,A -85,B 0,C 180,E1 -25907.427,E2 -25907.427} C_VEL
LIN {X 0,Y 121.255,Z 147.867,A -85,B 0,C 180,E1 -25908.461,E2 -25908.461} C_VEL
LIN {X 0,Y 121.914,Z 147.952,A -85,B 0,C 180,E1 -25918.772,E2 -25918.772} C_VEL
LIN {X 0,Y 122.667,Z 150.778,A -85,B 0,C 180,E1 -25922.268,E2 -25922.268} C_VEL
LIN {X 0,Y 124.819,Z 153.09,A -85,B 0,C 180,E1 -25927.289,E2 -25927.289} C_VEL
LIN {X 0,Y 126.082,Z 153.898,A -85,B 0,C 180,E1 -25929.434,E2 -25929.434} C_VEL
LIN {X 0,Y 127.671,Z 157.011,A -85,B 0,C 180,E1 -25932.125,E2 -25932.125} C_VEL
LIN {X 0,Y 130.214,Z 159.516,A -85,B 0,C 180,E1 -25935.386,E2 -25935.386} C_VEL
LIN {X 0,Y 132.584,Z 162.979,A -85,B 0,C 180,E1 -25938.14,E2 -25938.14} C_VEL
LIN {X 0,Y 133.71,Z 164.316,A -85,B 0,C 180,E1 -25939.288,E2 -25939.288} C_VEL
LIN {X 0,Y 137.327,Z 169.486,A -85,B 0,C 180,E1 -25942.682,E2 -25942.682} C_VEL
LIN {X 0,Y 140.86,Z 174.693,A -85,B 0,C 180,E1 -25945.56,E2 -25945.56} C_VEL
LIN {X 0,Y 144.745,Z 180.817,A -85,B 0,C 180,E1 -25948.376,E2 -25948.376} C_VEL
LIN {X 0,Y 149.428,Z 189.125,A -85,B 0,C 180,E1 -25951.455,E2 -25951.455} C_VEL
LIN {X 0,Y 154.239,Z 201.641,A -85,B 0,C 180,E1 -25954.526,E2 -25954.526} C_VEL
LIN {X 0,Y 157.081,Z 210.675,A -85,B 0,C 180,E1 -25956.29,E2 -25956.29} C_VEL
LIN {X 0,Y 152.477,Z 269.482,A -85,B 0,C 180,E1 -25958.551,E2 -25958.551} C_VEL
LIN {X 0,Y 150.308,Z 284.213,A -85,B 0,C 180,E1 -25959.518,E2 -25959.518} C_VEL
LIN {X 0,Y 147.425,Z 297.703,A -85,B 0,C 180,E1 -25960.824,E2 -25960.824} C_VEL
LIN {X 0,Y 143.444,Z 311.772,A -85,B 0,C 180,E1 -25962.706,E2 -25962.706} C_VEL
LIN {X 0,Y 139.154,Z 324.37,A -85,B 0,C 180,E1 -25965.009,E2 -25965.009} C_VEL
LIN {X 0,Y 135.698,Z 333.588,A -85,B 0,C 180,E1 -25967.211,E2 -25967.211} C_VEL
LIN {X 0,Y 132.355,Z 341.423,A -85,B 0,C 180,E1 -25969.429,E2 -25969.429} C_VEL
LIN {X 0,Y 127.928,Z 351.047,A -85,B 0,C 180,E1 -25972.827,E2 -25972.827} C_VEL
LIN {X 0,Y 123.35,Z 360.711,A -85,B 0,C 180,E1 -25977.236,E2 -25977.236} C_VEL
LIN {X 0,Y 119.05,Z 369.635,A -85,B 0,C 180,E1 -25982.573,E2 -25982.573} C_VEL
LIN {X 0,Y 116.506,Z 375.313,A -85,B 0,C 180,E1 -25986.92,E2 -25986.92} C_VEL
LIN {X 0,Y 114.262,Z 380.775,A -85,B 0,C 180,E1 -25992.094,E2 -25992.094} C_VEL
LIN {X 0,Y 112.647,Z 386.497,A -85,B 0,C 180,E1 -25999.218,E2 -25999.218} C_VEL
LIN {X 0,Y 112.266,Z 388.736,A -85,B 0,C 180,E1 -26002.813,E2 -26002.813} C_VEL
LIN {X 0,Y 112.145,Z 390.587,A -85,B 0,C 180,E1 -26006.412,E2 -26006.412} C_VEL
LIN {X 0,Y 112.28,Z 392.068,A -85,B 0,C 180,E1 -26010.005,E2 -26010.005} C_VEL
LIN {X 0,Y 112.211,Z 393.17,A -85,B 0,C 180,E1 -26013.596,E2 -26013.596} C_VEL
LIN {X 0,Y 112.708,Z 394.353,A -85,B 0,C 180,E1 -26020.787,E2 -26020.787} C_VEL
LIN {X 0,Y 114.567,Z 394.236,A -85,B 0,C 180,E1 -26027.867,E2 -26027.867} C_VEL
LIN {X 0,Y 118.351,Z 392.723,A -85,B 0,C 180,E1 -26034.927,E2 -26034.927} C_VEL
LIN {X 0,Y 119.643,Z 391.786,A -85,B 0,C 180,E1 -26037.661,E2 -26037.661} C_VEL
LIN {X 0,Y 120.618,Z 389.848,A -85,B 0,C 180,E1 -26042.286,E2 -26042.286} C_VEL
LIN {X 0,Y 122.3,Z 387.469,A -85,B 0,C 180,E1 -26046.755,E2 -26046.755} C_VEL
LIN {X 0,Y 124.607,Z 385.667,A -85,B 0,C 180,E1 -26049.133,E2 -26049.133} C_VEL
LIN {X 0,Y 131.985,Z 380.633,A -85,B 0,C 180,E1 -26053.813,E2 -26053.813} C_VEL
LIN {X 0,Y 138.717,Z 375.462,A -85,B 0,C 180,E1 -26057.282,E2 -26057.282} C_VEL
LIN {X 0,Y 147.255,Z 368.038,A -85,B 0,C 180,E1 -26060.861,E2 -26060.861} C_VEL
LIN {X 0,Y 154.943,Z 360.342,A -85,B 0,C 180,E1 -26063.622,E2 -26063.622} C_VEL
LIN {X 0,Y 162.956,Z 351.108,A -85,B 0,C 180,E1 -26066.127,E2 -26066.127} C_VEL
LIN {X 0,Y 171.376,Z 339.867,A -85,B 0,C 180,E1 -26068.32,E2 -26068.32} C_VEL
LIN {X 0,Y 178.51,Z 328.49,A -85,B 0,C 180,E1 -26070.02,E2 -26070.02} C_VEL
LIN {X 0,Y 185.183,Z 315.878,A -85,B 0,C 180,E1 -26071.364,E2 -26071.364} C_VEL
LIN {X 0,Y 190.394,Z 303.667,A -85,B 0,C 180,E1 -26072.369,E2 -26072.369} C_VEL
LIN {X 0,Y 194.943,Z 290.191,A -85,B 0,C 180,E1 -26073.167,E2 -26073.167} C_VEL
LIN {X 0,Y 198.347,Z 276.426,A -85,B 0,C 180,E1 -26073.744,E2 -26073.744} C_VEL
LIN {X 0,Y 200.495,Z 262.877,A -85,B 0,C 180,E1 -26074.147,E2 -26074.147} C_VEL
LIN {X 0,Y 201.808,Z 250.377,A -85,B 0,C 180,E1 -26074.464,E2 -26074.464} C_VEL
LIN {X 0,Y 200.814,Z 246.932,A -85,B 0,C 180,E1 -26075.746,E2 -26075.746} C_VEL
LIN {X 0,Y 198.723,Z 240.756,A -85,B 0,C 180,E1 -26078.701,E2 -26078.701} C_VEL
LIN {X 0,Y 196.795,Z 235.616,A -85,B 0,C 180,E1 -26082.188,E2 -26082.188} C_VEL
LIN {X 0,Y 195.601,Z 232.865,A -85,B 0,C 180,E1 -26085.1,E2 -26085.1} C_VEL
LIN {X 0,Y 194.429,Z 229.556,A -85,B 0,C 180,E1 -26091.68,E2 -26091.68} C_VEL
LIN {X 0,Y 194.547,Z 229.624,A -85,B 0,C 180,E1 -26094.202,E2 -26094.202} C_VEL
LIN {X 0,Y 196.033,Z 233.357,A -85,B 0,C 180,E1 -26100.365,E2 -26100.365} C_VEL
LIN {X 0,Y 197.595,Z 236.847,A -85,B 0,C 180,E1 -26103.662,E2 -26103.662} C_VEL
LIN {X 0,Y 199.557,Z 241.091,A -85,B 0,C 180,E1 -26106.685,E2 -26106.685} C_VEL
LIN {X 0,Y 202.152,Z 246.8,A -85,B 0,C 180,E1 -26109.846,E2 -26109.846} C_VEL
LIN {X 0,Y 199.704,Z 267.273,A -85,B 0,C 180,E1 -26110.383,E2 -26110.383} C_VEL
LIN {X 0,Y 196.666,Z 281.739,A -85,B 0,C 180,E1 -26110.957,E2 -26110.957} C_VEL
LIN {X 0,Y 192.871,Z 294.45,A -85,B 0,C 180,E1 -26111.667,E2 -26111.667} C_VEL
LIN {X 0,Y 188.194,Z 306.807,A -85,B 0,C 180,E1 -26112.665,E2 -26112.665} C_VEL
LIN {X 0,Y 182.527,Z 318.828,A -85,B 0,C 180,E1 -26113.924,E2 -26113.924} C_VEL
LIN {X 0,Y 175.955,Z 330.345,A -85,B 0,C 180,E1 -26115.495,E2 -26115.495} C_VEL
LIN {X 0,Y 168.5,Z 341.268,A -85,B 0,C 180,E1 -26117.418,E2 -26117.418} C_VEL
LIN {X 0,Y 160.569,Z 351.199,A -85,B 0,C 180,E1 -26119.763,E2 -26119.763} C_VEL
LIN {X 0,Y 152.248,Z 360.13,A -85,B 0,C 180,E1 -26122.588,E2 -26122.588} C_VEL
LIN {X 0,Y 143.372,Z 368.3,A -85,B 0,C 180,E1 -26126.168,E2 -26126.168} C_VEL
LIN {X 0,Y 134.585,Z 375.233,A -85,B 0,C 180,E1 -26130.493,E2 -26130.493} C_VEL
LIN {X 0,Y 127.962,Z 379.79,A -85,B 0,C 180,E1 -26134.522,E2 -26134.522} C_VEL
LIN {X 0,Y 120.177,Z 384.295,A -85,B 0,C 180,E1 -26140.507,E2 -26140.507} C_VEL
LIN {X 0,Y 113.872,Z 387.214,A -85,B 0,C 180,E1 -26147.235,E2 -26147.235} C_VEL
LIN {X 0,Y 109.155,Z 388.637,A -85,B 0,C 180,E1 -26154.581,E2 -26154.581} C_VEL
LIN {X 0,Y 106.146,Z 388.594,A -85,B 0,C 180,E1 -26162.383,E2 -26162.383} C_VEL
LIN {X 0,Y 104.812,Z 387.085,A -85,B 0,C 180,E1 -26170.406,E2 -26170.406} C_VEL
LIN {X 0,Y 104.715,Z 384.16,A -85,B 0,C 180,E1 -26178.379,E2 -26178.379} C_VEL
LIN {X 0,Y 105.794,Z 380.535,A -85,B 0,C 180,E1 -26185.014,E2 -26185.014} C_VEL
LIN {X 0,Y 107.706,Z 375.422,A -85,B 0,C 180,E1 -26191.864,E2 -26191.864} C_VEL
LIN {X 0,Y 110.637,Z 369.105,A -85,B 0,C 180,E1 -26198.212,E2 -26198.212} C_VEL
LIN {X 0,Y 114.685,Z 361.234,A -85,B 0,C 180,E1 -26204.184,E2 -26204.184} C_VEL
LIN {X 0,Y 119.067,Z 352.765,A -85,B 0,C 180,E1 -26209.09,E2 -26209.09} C_VEL
